	(* Reset Device by setting Error State  **********************)
	12:	
		IoDevReset(DEVICEID	:= DevId,RESET	:= TRUE );
		IF NOT IoDevReset.BUSY
		THEN
			IF IoDevReset.ERR THEN
				Busy										:= FALSE;
				Error										:= TRUE;
				ErrorId										:= IoDevReset.ERRID;
				ErrorText									:= CONCAT('IOF_DeviceReset Id: ',UDINT_TO_STRING(ErrorId));
				state 										:= 0;
			ELSE //Tr to                         					
				Error										:= FALSE;
				ErrorId										:= 0;
				ErrorText									:= '';
				DevResetDone 								:= TRUE;
				TON_TimeoutSetStatus(IN := FALSE);
				state 										:= 10;
			END_IF
		ELSE
			;
		END_IF
		
	(* Start to clear frame statistic **********************************)
	20: 
		FrameStatisticClearCRC(bExecute := Options.0);
		IF NOT FrameStatisticClearCRC.bBusy
		THEN
			IF FrameStatisticClearCRC.bError THEN
				Busy										:= FALSE;
				Error										:= TRUE;
				ErrorId										:= FrameStatisticClearCRC.nErrId;
				ErrorText									:= CONCAT('FB_EcMasterFrameStatisticClearCRC Id: ',UDINT_TO_STRING(ErrorId));
				state 										:= 0;
			ELSE                
				state 										:= state + 1;
			END_IF
		END_IF		
	
	21: 
		FrameStatisticClearFrames(bExecute := Options.1);
		IF NOT FrameStatisticClearFrames.bBusy
		THEN
			IF FrameStatisticClearFrames.bError THEN
				Busy										:= FALSE;
				Error										:= TRUE;
				ErrorId										:= FrameStatisticClearFrames.nErrId;
				ErrorText									:= CONCAT('FB_EcMasterFrameStatisticClearFrames Id: ',UDINT_TO_STRING(ErrorId));
				state 										:= 0;
			ELSE                
				state 										:= state + 1;
			END_IF
		END_IF	

	22: 
		FrameStatisticClearTxRxErr(bExecute := Options.2);
		IF NOT FrameStatisticClearTxRxErr.bBusy
		THEN
			IF FrameStatisticClearTxRxErr.bError THEN
				Busy										:= FALSE;
				Error										:= TRUE;
				ErrorId										:= FrameStatisticClearTxRxErr.nErrId;
				ErrorText									:= CONCAT('FB_EcMasterFrameStatisticClearTxRxErr Id: ',UDINT_TO_STRING(ErrorId));
				state 										:= 0;
			ELSE                
				Busy										:= FALSE;
				Done										:= TRUE;
				state 										:= 0;
			END_IF
		END_IF	
		
	ELSE
		;
	END_CASE
                										
(*********************************************************************)

{attribute 'monitoring' := 'call'}
PROPERTY PUBLIC optClearCRCErrorCounter : BOOL
GET
optClearCRCErrorCounter := Options.0;
END_GET
SET
Options.0 := optClearCRCErrorCounter;
END_SET
END_PROPERTY

{attribute 'monitoring' := 'call'}
PROPERTY PUBLIC optClearLostFramesCounter : BOOL
GET
optClearLostFramesCounter := Options.1;
END_GET
SET
Options.1 := optClearLostFramesCounter;
END_SET
END_PROPERTY

{attribute 'monitoring' := 'call'}
PROPERTY PUBLIC optClearTCRXErrCounter : BOOL
GET
optClearTCRXErrCounter := Options.2;
END_GET
SET
Options.2 := optClearTCRXErrCounter;
END_SET
END_PROPERTY

{attribute 'monitoring' := 'call'}
PROPERTY PUBLIC optForceDevReset : BOOL
GET
optForceDevReset := Options.7;
END_GET
SET
Options.7 := optForceDevReset;
END_SET
END_PROPERTY

END_FUNCTION_BLOCK

// POUs/Fieldbus/EtherCAT/_Components/EcSlavesDiag
{attribute 'no_check'}
{attribute 'enable_dynamic_creation'}
FUNCTION_BLOCK EcSlavesDiag EXTENDS FbBase
VAR CONSTANT
	SLAVE_ADDR_OFFSET										:	UINT := 1000;
	DEL_SSTATE_CHANGED										:	 TIME := T#2S;
END_VAR
VAR_OUTPUT CONSTANT         								
	MIN_SLAVES												: 	UINT := 1;
	MAX_SLAVES												: 	UINT := PARAM.ETHERCAT_DIAG_MAX_SLAVES;	//EC_MAX_SLAVES = 65535 Slaves;
	
{attribute 'displaymode':='binary'}
	OPTION_READ_SCAN_SLAVES									:	BYTE := 2#0000_0001; //Read scanned slaves identity and link State
{attribute 'displaymode':='binary'}
	OPTION_SORT_INFO_DATA									:	BYTE := 2#0000_0010; //Sort list of slaves InfoData according to scanned/physical sequence
{attribute 'displaymode':='binary'}
	OPTION_UPDATE_TOPO_DATA									:	BYTE := 2#0000_0100; //Read topology data, helpful if hot connect groups are configured
{attribute 'displaymode':='binary'}
	OPTION_UPDATE_CONFIG_DATA								:	BYTE := 2#0000_1000; //Read info slave data with with every execution	
END_VAR           
VAR_INPUT
	MasterAmsNetId											:	T_AmsNetId;
{attribute 'displaymode':='binary'}
	Options													:	BYTE := 0;
END_VAR
VAR_OUTPUT         
	NoOfSlaves												:	UINT;			//shows number of configured 
	NoOfSlavesNOK											:	UINT;  			//Shows number of slaves not in OP or with CRC error etc
	NoOfHCGroups											:	UINT;  			//Shows number of hot connect groups
	NoOfHCSlaves											:	UINT;  			//Shows number of slave in a hot connect group
	InfoData												:	ARRAY [MIN_SLAVES..MAX_SLAVES] OF EC_SLAVE_DIAG_INFO_DATA; //configures slaves			
	LastActiveSlave											:	EC_SLAVE_DIAG_INFO_DATA;	//shows last slave in OP connected to port A 
	FirstErrorSlave											:	EC_SLAVE_DIAG_INFO_DATA;	//shows first slave with an error
	InfoDataSorted											:	BOOL; //Info data list sorted according physical sequence vs. configured seq.
	InvalidVPRS												:	BOOL; //Invalid VPRS active
	ErrorText												:	STRING;		//shows error text of FB
	ExecutionTime											: 	TIME; //Total cycle time to execute the FB
END_VAR                     								         								
VAR                         								
(* Cache ********************************************************)               								
	pMemory													:	POINTER TO BYTE;
	SizeOfMemory											:	UDINT;
	MemNoOfSlaves											:	UINT;	
	ScannedSeqMixed											:	BOOL; //Scanned slave sequence is different to configured 

	pScannedSlaves											:	POINTER TO ARRAY [MIN_SLAVES..MAX_SLAVES] OF Tc2_EtherCAT.ST_EcSlaveScannedData;
	pConfigSlaves											:	POINTER TO ARRAY [MIN_SLAVES..MAX_SLAVES] OF Tc2_EtherCAT.ST_EcSlaveConfigData; 
	pSlavesState											:	POINTER TO ARRAY [MIN_SLAVES..MAX_SLAVES] OF Tc2_EtherCAT.ST_EcSlaveState;
	pSlavesStatusCode										:	POINTER TO ARRAY [MIN_SLAVES..MAX_SLAVES] OF DWORD;
	pTopologyData											:	POINTER TO ARRAY [MIN_SLAVES..MAX_SLAVES] OF Tc2_EtherCAT.ST_TopologyDataEx;
	
	StartTime												:	TIME;
	
(* timer ********************************************************)

(* trigger ********************************************************)

(* function-blocks *************************************************)
	EcGetSlaveCount											:	FB_EcGetSlaveCount := (tTimeout	:= T#60S);
	EcGetConfSlaves											:	FB_EcGetConfSlaves := (tTimeout	:= T#60S);
	EcGetScannedSlaves										:	FB_EcGetScannedSlaves := (tTimeout	:= T#60S);
	EcGetAllSlaveStateS										:	FB_EcGetAllSlaveStateS := (tTimeout	:= T#60S);
	EcGetAllSlaveCrcErrors									:	FB_EcGetAllSlaveCrcErrors := (tTimeout	:= T#60S);
	EcGetAllSlaveAbnormalStateChanges						:	FB_EcGetAllSlaveAbnormalStateChanges := (tTimeout	:= T#60S);	
	EcGetSlaveTopologyInfo									: 	FB_EcGetSlaveTopologyInfo := (tTimeout	:= T#60S);	
	
(* dummy **********************************************************)
	i,k,idx													:	UINT := 0;
	
END_VAR

	(* Check EtherCAT slaves status			V1	*)
	(********************************************)

(* Sequence *********************************)
	rtExecute(CLK := Execute);

	CASE State OF
	0:
		Busy 												:= FALSE;
		IF rtExecute.Q
		THEN //Clear data if FB is disabled or started
			Busy 											:= TRUE;
			Done											:= FALSE;
			Error											:= FALSE;
			Errorid											:= 0;
			ErrorText										:= '';	

		//	NoOfSlavesNIO									:= 0;	
			InvalidVPRS										:= FALSE;
			ScannedSeqMixed									:= FALSE;

			StartTime										:= TIME();
			ExecutionTime									:= T#0MS;
			
			EcGetSlaveCount(bExecute := FALSE,sNetId := MasterAmsNetId);
			EcGetConfSlaves(bExecute := FALSE,sNetId := MasterAmsNetId);
			EcGetSlaveTopologyInfo(bExecute := FALSE,sNetId := MasterAmsNetId);
			EcGetAllSlaveStates(bExecute := FALSE, sNetId := MasterAmsNetId);
			EcGetAllSlaveCrcErrors(bExecute := FALSE,sNetId := MasterAmsNetId);
			EcGetAllSlaveAbnormalStateChanges(bExecute := FALSE,sNetId := MasterAmsNetId);
			EcGetScannedSlaves(bExecute := FALSE,sNetId := MasterAmsNetId);
			
			MEMSET(ADR(LastActiveSlave),0,SIZEOF(LastActiveSlave));
			MEMSET(ADR(FirstErrorSlave),0,SIZEOF(FirstErrorSlave));
			
			IF NoOfSlaves = 0
			THEN
				State										:= 1;
			ELSIF Options.3 OR EcGetConfSlaves.nTotalSlaves = 0 OR InfoDataSorted
			THEN //Read config it not done or enabled
				State										:= 2;
			ELSIF Options.2 OR EcGetSlaveTopologyInfo.nSlaves = 0 OR InfoDataSorted
			THEN
				State										:= 10;
			ELSE
				State										:= 20;
			END_IF
		ELSIF NOT Execute
		THEN
			Done											:= FALSE;
			Error											:= FALSE;
			Errorid											:= 0;
			ErrorText										:= '';	
		END_IF
		IF StartTime > T#0MS AND ExecutionTime = T#0MS
		THEN
			ExecutionTime									:= TIME() - StartTime;
		END_IF
	
	(* Read no of configured slaves *********************************************************************)
	1:
		EcGetSlaveCount(bExecute := NoOfSlaves = 0);
		IF NOT EcGetSlaveCount.bBusy
		THEN
			IF EcGetSlaveCount.bError 
			THEN
				Busy										:= FALSE;
				Error										:= TRUE;
				ErrorId										:= EcGetSlaveCount.nErrId;
				ErrorText									:= CONCAT('EcGetSlaveCount Id: ',UDINT_TO_STRING(ErrorId));
				State 										:= 0;
			ELSIF EcGetSlaveCount.bExecute AND NoOfSlaves <> EcGetSlaveCount.nSlaves
			THEN
				NoOfSlaves									:= EcGetSlaveCount.nSlaves;					

				//Init Info Data 	
				MEMSET(ADR(InfoData),0,SIZEOF(InfoData));

				k 											:= NoOfSlaves + 1;
				//Set buffer lenght according to needed memory space
				EcGetConfSlaves.cbBufLen					:= SIZEOF(Tc2_EtherCAT.ST_EcSlaveConfigData) * k;
				EcGetScannedSlaves.cbBufLen					:= SIZEOF(Tc2_EtherCAT.ST_EcSlaveScannedData) * k;
				EcGetAllSlaveStates.cbBufLen				:= SIZEOF(Tc2_EtherCAT.ST_EcSlaveState) * k;
				EcGetAllSlaveCrcErrors.cbBufLen				:= SIZEOF(DWORD) * k;	
				EcGetSlaveTopologyInfo.cbBufLen				:= SIZEOF(Tc2_EtherCAT.ST_TopologyDataEx) * k;	
				EcGetAllSlaveAbnormalStateChanges.cbBufLen	:= EcGetAllSlaveCrcErrors.cbBufLen;						
					
				//Allocate dynamic buffer memory 
				IF Allocate(MAX(EcGetSlaveTopologyInfo.cbBufLen,MAX(MAX(EcGetConfSlaves.cbBufLen,EcGetAllSlaveCrcErrors.cbBufLen), MAX(EcGetScannedSlaves.cbBufLen,EcGetAllSlaveStateS.cbBufLen) )))
				THEN
					//Write buffer lenght per FB	
					pConfigSlaves							:= pMemory;
					pScannedSlaves							:= pMemory;
					pSlavesState							:= pMemory;
					pSlavesStatusCode						:= pMemory;	
					pTopologyData							:= pMemory;	
					
					State 									:= State + 1;			
				ELSE
					Busy									:= FALSE;
					Error									:= TRUE;
					ErrorId									:= E_AdsErr.DEVICE_NOMEMORY; //No memory
					ErrorText								:= CONCAT('EcSlavesDiag.allocate() Id: ',UDINT_TO_STRING(ErrorId));
					State 									:= 0;	
				END_IF

			ELSE
				State 										:= State + 1;
			END_IF
		ELSE
			;
		END_IF		
	
	
	(* Read slaves "configuration" ************************************************************************************************************)
	2:
		EcGetConfSlaves(bExecute := TRUE, pArrEcConfSlaveInfo := pConfigSlaves, cbBufLen := (* See State 1 *) );
			
		IF NOT EcGetConfSlaves.bBusy
		THEN
			IF EcGetConfSlaves.bError 
			THEN
				Busy										:= FALSE;
				Error										:= TRUE;
				ErrorId										:= EcGetConfSlaves.nErrorId;
				ErrorText									:= CONCAT('FB_EcGetConfSlaves Id: ',UDINT_TO_STRING(ErrorId));
				State										:= 0;     
					
			ELSIF EcGetConfSlaves.nSlaves > MAX_SLAVES
			THEN
				Busy										:= FALSE;
				Error										:= TRUE;
				ErrorId										:= E_AdsErr.DEVICE_INVALIDSIZE  ;
				ErrorText									:= CONCAT('No of config slaves > PARAM.ETHERCAT_MASTER_DIAG_MAX_SLAVES, please update value to ', TO_STRING(EcGetConfSlaves.nSlaves));
				State										:= 0;  					
			ELSE
				State 										:= State + 1;
			END_IF
		END_IF	
		
		
	3: //Fill structure	
		k													:= MIN(EcGetConfSlaves.nSlaves, NoOfSlaves);
		FOR i := MIN_SLAVES TO k DO
			InfoData[i].Addr								:= pConfigSlaves^[i].nAddr;
			InfoData[i].ConfigType							:= pConfigSlaves^[i].sType; 
		//	InfoData[i].DevType								:= pConfigSlaves^[i].nDevType;
			InfoData[i].ConfigName							:= DELETE(pConfigSlaves^[i].sName, LEN(InfoData[i].ConfigType) + 3 , FIND(pConfigSlaves^[i].sName,InfoData[i].ConfigType) - 1); //Delete type if in brakets 	
			InfoData[i].ConfigTypeIdentity					:= F_ConvProductCodeToString(pConfigSlaves^[i].stSlaveIdentity);
			InfoData[i].ConfigIdentity						:= pConfigSlaves^[i].stSlaveIdentity;
		//	InfoData[i].LinkState							:= pConfigSlaves^[i].nLinkStatus; see read slaves state					
		END_FOR
		
		State 												:= SEL(Options.2 OR EcGetSlaveTopologyInfo.nSlaves = 0 OR InfoDataSorted, 20, 10);	
		
	(* Read slaves "topology" information *******************************************************************************************************)
	10:
		EcGetSlaveTopologyInfo(bExecute := NoOfSlaves > 0 , sNetId	:= MasterAmsNetId,  pAddrBuf := pTopologyData,  cbBufLen	:= (* See State 1 *));
		IF NOT EcGetSlaveTopologyInfo.bBusy
		THEN
			IF EcGetSlaveTopologyInfo.bError 
			THEN
				Busy										:= FALSE;
				Error										:= TRUE;
				ErrorId										:= EcGetSlaveTopologyInfo.nErrId;
				ErrorText									:= CONCAT('EcGetSlaveTopologyInfo Id: ',UDINT_TO_STRING(ErrorId));
				State 										:= 0;
			ELSIF EcGetSlaveTopologyInfo.nSlaves > MAX_SLAVES
			THEN
				Busy										:= FALSE;
				Error										:= TRUE;
				ErrorId										:= E_AdsErr.DEVICE_INVALIDSIZE  ;
				ErrorText									:= CONCAT('No of scanned slaves > PARAM.ETHERCAT_MASTER_DIAG_MAX_SLAVES, please update value to ', TO_STRING(EcGetScannedSlaves.nSlaves));
				State										:= 0;  	
			ELSE
				State 										:= State + 1;
			END_IF
		ELSE
			;
		END_IF	

	11:	//Fill structure		
		NoOfHCGroups										:= 0;
		NoOfHCSlaves										:= 0;
		k													:= MIN(EcGetSlaveTopologyInfo.nSlaves, NoOfSlaves);
		FOR i := MIN_SLAVES TO k DO                 		
			InfoData[i].TopoOwnPhysicalAddr					:= pTopologyData^[i].nOwnPhysicalAddr; 
			InfoData[i].TopologyStatus						:= pTopologyData^[i].nStatusBits;
			InfoData[i].HCSlaveCountCfg  					:= pTopologyData^[i].nHCSlaveCountCfg;
			InfoData[i].HCSlaveCountAct  					:= pTopologyData^[i].nHCSlaveCountAct;
			InfoData[i].AutoIncAddr   						:= pTopologyData^[i].nOwnAutoIncAddr;
			InfoData[i].PhysicalPortAddr    				:= pTopologyData^[i].stPhysicalAddr;
			InfoData[i].AutoIncPortAddr    					:= pTopologyData^[i].stAutoIncAddr;
			                                        		
			InfoData[i].HotConnectNodeStart 				:= InfoData[i].TopologyStatus.3;
			InfoData[i].HotConnectSlave 					:= InfoData[i].TopologyStatus.4;
                                                    		
			NoOfHCGroups									:= SEL(InfoData[i].HotConnectNodeStart , NoOfHCGroups, NoOfHCGroups + 1);
			NoOfHCSlaves									:= SEL(InfoData[i].HotConnectSlave , NoOfHCSlaves, NoOfHCSlaves + 1);
			                                        	
		END_FOR				                        	
		State 												:= 20;
		
	(* Read slaves "EtherCAT State and link state" ***************************************************************************************)
	20	:
		EcGetAllSlaveStateS(bExecute := NoOfSlaves > 0, pStateBuf:=  pSlavesState, cbBufLen	:= (* See State 1 *));
					
		IF NOT EcGetAllSlaveStateS.bBusy
		THEN
			IF EcGetAllSlaveStateS.bError 
			THEN
				Busy										:= FALSE;
				Error										:= TRUE;
				ErrorId										:= EcGetAllSlaveStateS.nErrId;
				ErrorText									:= CONCAT('FB_EcGetAllSlaveStates Id: ',UDINT_TO_STRING(ErrorId));
				State 										:= 0;
			ELSE
				k											:= MIN(EcGetAllSlaveStateS.nSlaves, NoOfSlaves);
				FOR i := MIN_SLAVES TO k DO
					InfoData[i].LinkState					:= pSlavesState^[i].linkState;
					InfoData[i].DevState					:= pSlavesState^[i].deviceState;
					InfoData[i].DevStateText				:= F_ConvSlaveStateToString(pSlavesState^[i]);
					InfoData[i].DevStateBits				:= F_ConvSlaveStateToBitsEx(pSlavesState^[i]);	
					InfoData[i].ErrorIdentCode.0			:= InfoData[i].DevStateBits.bInvVPRS; //Wrong slave
					IF InfoData[i].ErrorIdentCode.0 THEN InvalidVPRS := TRUE; END_IF
					InfoData[i].ErrorIdentCode.1			:= NOT InfoData[i].ErrorIdentCode.0 AND NOT InfoData[i].DevStateBits.bOp AND_THEN(NOT InfoData[i].HotConnectSlave OR NOT InfoData[i].DevStateBits.bInit); //Wrong State
				END_FOR	

				State 										:= State + 1;
			END_IF
		ELSE
			;
		END_IF	
		
	(* Get all slaves "CRC counter" ********************************************************************)
	21:	
		EcGetAllSlaveCrcErrors(bExecute := NoOfSlaves > 0, sNetId	:= MasterAmsNetId,  pCrcErrorBuf:= pSlavesStatusCode,  cbBufLen	:= (* See State 1 *));
		IF NOT EcGetAllSlaveCrcErrors.bBusy
		THEN
			IF EcGetAllSlaveCrcErrors.bError 
			THEN
				Busy										:= FALSE;
				Error										:= TRUE;
				ErrorId										:= EcGetAllSlaveStateS.nErrId;
				ErrorText									:= CONCAT('FB_EcGetAllSlaveCrcErrors Id: ',UDINT_TO_STRING(ErrorId));
				State 										:= 0;
			ELSE
				k											:= MIN(EcGetAllSlaveCrcErrors.nSlaves, NoOfSlaves);
				FOR i := MIN_SLAVES TO k DO
					InfoData[i].ErrorIdentCode.2			:= InfoData[i].CntOfCRCErrors <> pSlavesStatusCode^[i] AND pSlavesStatusCode^[i] > 0; //CRC error increased
					InfoData[i].CntOfCRCErrors				:= pSlavesStatusCode^[i];				
				END_FOR				
				
				State 										:= State + 1;
			END_IF
		ELSE
			;
		END_IF
		
	(* Get all slaves "no of abnormal state change" *****************************************************************************)
	22:	
		EcGetAllSlaveAbnormalStateChanges(bExecute := NoOfSlaves > 0, sNetId	:= MasterAmsNetId,  pAddrBuf := pSlavesStatusCode,  cbBufLen	:= (* See State 1 *));
		IF NOT EcGetAllSlaveAbnormalStateChanges.bBusy
		THEN
			IF EcGetAllSlaveAbnormalStateChanges.bError 
			THEN
				Busy										:= FALSE;
				Error										:= TRUE;
				ErrorId										:= EcGetAllSlaveAbnormalStateChanges.nErrId;
				ErrorText									:= CONCAT('FB_EcGetAllSlaveAbnormalStateChanges Id: ',UDINT_TO_STRING(ErrorId));
				State 										:= 0;
			ELSE
				k											:= MIN(EcGetAllSlaveAbnormalStateChanges.nSlaves, NoOfSlaves);
				FOR i := MIN_SLAVES TO k DO
					InfoData[i].ErrorIdentCode.3			:= InfoData[i].NoOfAbnormalStateChanges <> pSlavesStatusCode^[i] AND pSlavesStatusCode^[i] > 0; //Abnormal State change increased
					InfoData[i].NoOfAbnormalStateChanges	:= pSlavesStatusCode^[i];	
				END_FOR				
				
				State 										:= SEL(Options.0 OR EcGetScannedSlaves.nSlaves = 0, 40, 30);
			END_IF
		ELSE
			;
		END_IF

	(* Start to read scanned slaves *************************************************************************)
	30:
		EcGetScannedSlaves(bExecute := TRUE, pArrEcScannedSlaveInfo  := pScannedSlaves, cbBufLen := (* See State 1 *));
			
		IF NOT EcGetScannedSlaves.bBusy
		THEN
			IF EcGetScannedSlaves.bError 
				AND EcGetScannedSlaves.nErrorId <> 1817 //device has a timeout -> not error if no slave is connected 
			THEN
				Busy										:= FALSE;
				Error										:= TRUE;
				ErrorId										:= EcGetScannedSlaves.nErrorId;
				ErrorText									:= CONCAT('FB_EcGetScannedSlaves Id: ',UDINT_TO_STRING(ErrorId));
				State										:= 0;     

			ELSIF EcGetScannedSlaves.nSlaves > MAX_SLAVES
			THEN
				Busy										:= FALSE;
				Error										:= TRUE;
				ErrorId										:= E_AdsErr.DEVICE_INVALIDSIZE  ;
				ErrorText									:= CONCAT('No of scanned slaves > PARAM.ETHERCAT_MASTER_DIAG_MAX_SLAVES, please update value to ', TO_STRING(EcGetScannedSlaves.nSlaves));
				State										:= 0;  			
			
			ELSE	
				FOR i := MIN_SLAVES TO NoOfSlaves 
				DO					
					InfoData[i].ScannedTypeIdentity			:= '<not present>';
					MEMSET(ADR(InfoData[i].ScannedIdentity),0,SIZEOF(InfoData[i].ScannedIdentity));								
					InfoData[i].DataLinkStatusReg			:= 0;	
					InfoData[i].ScannedSeq					:= 0;						
				END_FOR
				State 										:= SEL(EcGetScannedSlaves.nSlaves = 0, State + 1, 40);
			END_IF
		END_IF
		
	31: //Fill structure
		k													:= MIN(EcGetScannedSlaves.nSlaves,NoOfSlaves); //No of scanned slaves
		idx													:= 0;
		ScannedSeqMixed										:= FALSE;
		FOR i := MIN_SLAVES TO NoOfSlaves DO		
			IF i <= EcGetScannedSlaves.nSlaves
			THEN
				idx											:= SEL(pScannedSlaves^[i].nAddr > SLAVE_ADDR_OFFSET, idx + 1 ,pScannedSlaves^[i].nAddr - SLAVE_ADDR_OFFSET);
				InfoData[idx].ScannedTypeIdentity			:= F_ConvProductCodeToString(pScannedSlaves^[i].stSlaveIdentity);
				InfoData[idx].ScannedIdentity				:= pScannedSlaves^[i].stSlaveIdentity;				
				InfoData[idx].DataLinkStatusReg				:= pScannedSlaves^[i].ndlStatusReg;		
				InfoData[idx].ScannedSeq					:= i;	
				ScannedSeqMixed								:= i <> idx OR ScannedSeqMixed;
			ELSE
				EXIT;
			END_IF
		
		END_FOR
		
		State 												:= 40;
		
	(* Search for error slaves **************************************************************************)
	40:
		k													:= EcGetScannedSlaves.nSlaves + 1; 
		NoOfSlavesNOK										:= 0;
		FOR i := MIN_SLAVES TO NoOfSlaves				
		DO
			//Fill PhysicalSeq number of missed slaves for possible sorting
			IF ScannedSeqMixed AND Options.1
			THEN
				IF InfoData[i].ScannedSeq = 0
				THEN 										
					InfoData[i].ScannedSeq 					:= k;
					k										:= k + 1;
				END_IF
			END_IF
		
			//Search for first slave with error
			IF InfoData[i].ErrorIdentCode <> 0
			THEN
				NoOfSlavesNOK								:= NoOfSlavesNOK + 1;
				IF FirstErrorSlave.Addr = 0
				THEN
					FirstErrorSlave 						:= InfoData[i]; 					
					IF i - 1 > 0
					THEN
						LastActiveSlave 					:= InfoData[i - 1];
					END_IF
				END_IF						
			END_IF
		END_FOR   	
	
		IF ScannedSeqMixed AND Options.1
		THEN
			InfoDataSorted									:= TRUE;
			State											:= State + 1;
		ELSE
			InfoDataSorted									:= FALSE;
			Busy											:= FALSE;
			Done											:= TRUE;
			State											:= 0;   
		END_IF
	
	(* Sort InfoData list if sequence is mixed and option selected **************************************************************************)	
	41: 
		IF sortList()
		THEN
			Busy											:= FALSE;
			Done											:= TRUE;
			State											:= 0;   
		ELSE
			Busy											:= FALSE;
			Error											:= TRUE;
			ErrorId											:= E_AdsErr.DEVICE_INVALIDDATA  ; //Invalid data
			ErrorText										:= 'Error sorting InfoData list ';
			State											:= 0;  			
		END_IF	
 
	ELSE
		;
	END_CASE

(***********************************************************************)

METHOD PROTECTED FINAL allocate : BOOL
VAR_INPUT 
	MemSize													:	UDINT;
END_VAR
VAR
END_VAR
IF MemSize = 0
THEN
	allocate												:= FALSE;	
ELSIF pMemory = 0 
THEN
	pMemory													:= __NEW(BYTE,MemSize );
	SizeOfMemory											:= MemSize;
	IF PARAM.ENABLE_DEBUG_MSG_DYNAMIC_MEM_ALLOCATION
	THEN
		AdsLogHint('EngineeringToolbox | FB EcSlavesDiag | An instance allocated %s bytes from the dynamic memory of the ADS router memory pool', TO_STRING(MemSize));
	END_IF
	Allocate												:= TRUE;	
ELSIF MemSize > SizeOfMemory
THEN//Size increased, allocate new memory
	__DELETE(pMemory);  //Delete reference to old memory
	
	pMemory													:= __NEW(BYTE,MemSize );
	SizeOfMemory											:= MemSize;
	IF PARAM.ENABLE_DEBUG_MSG_DYNAMIC_MEM_ALLOCATION
	THEN
		AdsLogWarn('EngineeringToolbox | FB EcSlavesDiag | No of slaves increased and one instance allocated additional %s bytes from the dynamic memory of the ADS router memory pool', TO_STRING(MemSize));
	END_IF

	Allocate												:= TRUE;
ELSE
	Allocate												:= FALSE;
END_IF
END_METHOD

METHOD FB_exit : BOOL
VAR_INPUT
	bInCopyCode : BOOL; // if TRUE, the exit method is called for exiting an instance that is copied afterwards (online change).
END_VAR
IF NOT bInCopyCode AND pMemory <> 0
THEN //Release memory in case the PLC stopps
	__DELETE(pMemory);
	SizeOfMemory								:= 0;
END_IF
END_METHOD

{attribute 'monitoring' := 'call'}
PROPERTY PUBLIC optReadScannedSlaves : bool
GET
optReadScannedSlaves := Options.0;
END_GET
SET
OPtions.0 := optReadScannedSlaves;
END_SET
END_PROPERTY

{attribute 'monitoring' := 'call'}
PROPERTY PUBLIC optSortInfoData : bool
GET
optSortInfoData := Options.2;
END_GET
SET
OPtions.2 := optSortInfoData;
END_SET
END_PROPERTY

{attribute 'monitoring' := 'call'}
PROPERTY PUBLIC optUpdateConfigData : bool
GET
optUpdateConfigData := Options.3;
END_GET
SET
OPtions.3 := optUpdateConfigData;
END_SET
END_PROPERTY

{attribute 'monitoring' := 'call'}
PROPERTY PUBLIC optUpdateTopoData : bool
GET
optReadScannedSlaves := Options.1;
END_GET
SET
OPtions.1 := optReadScannedSlaves;
END_SET
END_PROPERTY

METHOD INTERNAL sortList : BOOL
VAR_INPUT
END_VAR
VAR
	SlaveInfoData1											:	EC_SLAVE_DIAG_INFO_DATA;
	SlaveInfoData2											:	EC_SLAVE_DIAG_INFO_DATA;
END_VAR
	sortList												:= TRUE;
	
	i														:= MIN_SLAVES;
	WHILE i <= NoOfSlaves OR SlaveInfoData1.ScannedSeq <> 0 
	DO
		IF SlaveInfoData1.ScannedSeq > 0
		THEN
			IF SlaveInfoData1.ScannedSeq > NoOfSlaves
			THEN //Error seq no
				sortList									:= FALSE;
				EXIT;
			ELSE
				SlaveInfoData2 								:= InfoData[SlaveInfoData1.ScannedSeq]; //Backup target
				InfoData[SlaveInfoData1.ScannedSeq].ScannedSeq	:= 0; //Mark as copied				
				InfoData[SlaveInfoData1.ScannedSeq]			:= SlaveInfoData1; //Copy from cache into target	
				SlaveInfoData1								:= SlaveInfoData2; //Write backed up data into cache
			END_IF

		ELSIF InfoData[i].ScannedSeq > 0 AND InfoData[i].ScannedSeq <> i
		THEN
			//Put target into cache
			SlaveInfoData1									:= InfoData[InfoData[i].ScannedSeq];
			InfoData[InfoData[i].ScannedSeq]				:= InfoData[i];		
			InfoData[i].ScannedSeq							:= 0; //Mark as copied
		ELSE
			;				
		END_IF   
		i													:= i + 1;
	END_WHILE;
END_METHOD

END_FUNCTION_BLOCK

// POUs/Fieldbus/EtherCAT/_Components/EcSlaveSupervisor
{attribute 'no_check'}
(* Set EtherCAT state(ReqState <> 0) or read state and CRC error counter of EtherCAT slave *)
FUNCTION_BLOCK EcSlaveSupervisor Extends FbBase
VAR_INPUT
	EcMasterAmsNetId										:	T_AmsNetId;
	SlaveAddr												: 	UINT; 		//-> Slave Port number!
{attribute 'displaymode':='hex'}
	ReqState												:	WORD := 0; (* 	EC_DEVICE_STATE_INIT		:BYTE 	:=16#01;
																				EC_DEVICE_STATE_PREOP		:BYTE 	:=16#02;
																				EC_DEVICE_STATE_BOOTSTRAP	:BYTE 	:=16#03;
																				EC_DEVICE_STATE_SAFEOP		:BYTE 	:=16#04;
																				EC_DEVICE_STATE_OP			:BYTE 	:=16#08; *)																				
END_VAR                     							
VAR_OUTPUT                  							
{attribute 'displaymode':='hex'}
	CurrState												: 	BYTE;	(* Shows current state 																					
																				EC_DEVICE_STATE_INIT		:BYTE 	:=16#01;
																				EC_DEVICE_STATE_PREOP		:BYTE 	:=16#02;
																				EC_DEVICE_STATE_BOOTSTRAP	:BYTE 	:=16#03;
																				EC_DEVICE_STATE_SAFEOP		:BYTE 	:=16#04;
																				EC_DEVICE_STATE_OP			:BYTE 	:=16#08; *)
{attribute 'displaymode':='hex'}
	linkState												: 	BYTE;	(* Shows state of link
																				EC_LINK_STATE_OK :BYTE :=16#00;
																				EC_LINK_STATE_NOT_PRESENT :BYTE :=16#01;
																				EC_LINK_STATE_LINK_WITHOUT_COMM :BYTE :=16#02;
																				EC_LINK_STATE_MISSING_LINK :BYTE :=16#04;
																				EC_LINK_STATE_ADDITIONAL_LINK :BYTE :=16#08;
																				EC_LINK_STATE_PORT_A :BYTE :=16#10;
																				EC_LINK_STATE_PORT_B :BYTE :=16#20;
																				EC_LINK_STATE_PORT_C :BYTE :=16#40;
																				EC_LINK_STATE_PORT_D :BYTE :=16#80; *)
																				
	ReqStateOK												:	BOOL;		//Requested state of slave is OK
	StateBits												:	ST_EcSlaveStateBitsEx;
	StateText												:	STRING(80);	//State as text
	CrcError    											:    ST_EcCrcErrorEx; (*Crc error of the EtherCAT slave device*)
END_VAR                 								
VAR                     								
	TON_GetStateTrig										:	TON;
	SetSlaveState											:	FB_EcSetSlaveSTATE := (tTimeout := DEFAULT_ADS_TIMEOUT);
	GetSlaveState											:	FB_EcGetSlaveSTATE := (tTimeout := DEFAULT_ADS_TIMEOUT);
	GetSlaveCrcErrorEx 										:	FB_EcGetSlaveCrcErrorEx  := (tTimeout := DEFAULT_ADS_TIMEOUT);
	MemReqState												:	WORD;
	ErrorText												:	STRING(40);
END_VAR

	(* Set EtherCAT state(ReqState <> 0) or read state and CRC error counter of EtherCAT slave *)
	(*******************************************************************************************)

(* Process ******************************************************)
	rtExecute(CLK := Execute);

	CASE state OF
	(* cyclic reading of state ***********************************)
	0:
		Busy 												:= FALSE;

		IF rtExecute.Q 
		THEN
			Busy 											:= TRUE;
			Done											:= FALSE;
			Error											:= FALSE;
			ErrorID											:= 0;
			Errortext										:= '';
			CurrState										:= 0;
			linkState										:= 0;
			ReqStateOK										:= FALSE;
			MEMSET(ADR(StateBits),0,SIZEOF(StateBits));
			MEMSET(ADR(CrcError),0,SIZEOF(CrcError));	
			StateText										:= '';
	
			SetSlaveSTATE(bExecute := FALSE, sNetId:= EcMasterAmsNetId,nSlaveAddr:= SlaveAddr);
			GetSlaveSTATE(bExecute := FALSE,sNetId:= EcMasterAmsNetId,nSlaveAddr:= SlaveAddr);
			GetSlaveCrcErrorEx(bExecute := FALSE,sNetId:= EcMasterAmsNetId,nSlaveAddr:= SlaveAddr);

			IF(ReqState <> CurrState
				OR ReqState <> MemReqState)
				AND ReqState <> 0
			THEN
				SetSlaveState(bExecute:= TRUE,reqState:= ReqState);
				MemReqState 								:= ReqState;
				state 										:= 10;

			ELSE
				(* Start Reading State *)
				GetSlaveState(bExecute	:= TRUE);
				state 										:= 1;
			END_IF

		ELSIF NOT Execute 
		THEN
			Done 											:= FALSE;
			Error											:= FALSE;
			ErrorID											:= 0;
			ErrorText										:= '';
		END_IF

	(* Read Slave State **************************************)
	1:
		(* Work block *)
		GetSlaveState();

		IF NOT GetSlaveState.bBusy
		THEN
			IF GetSlaveState.bError THEN
				Busy										:= FALSE;
				Error										:= TRUE;
				ErrorId										:= GetSlaveState.nErrId;
				ErrorText									:= CONCAT('FB_EcGetSlaveSTATE Id: ',UDINT_TO_STRING(ErrorId));
				state 										:= 0;
			ELSE       
				ReqStateOK 									:= (ReqState = CurrState OR ReqState = 0);         					
				CurrState 									:= GetSlaveState.state.deviceState;
				linkState 									:= GetSlaveState.State.linkState;
				StateText 									:= F_ConvStateToString(GetSlaveState.State.deviceState);
			 	StateBits							 		:= F_ConvSlaveStateToBitsEx(GetSlaveState.state);
				state										:= state + 1;
			END_IF
			GetSlaveSTATE(bExecute := FALSE);
		ELSE
			;
		END_IF

	(* Read Slave CRC Error Counter  **************************************)		
	2: 
		(* Work block *)
		GetSlaveCrcErrorEx();

		IF NOT GetSlaveCrcErrorEx.bBusy
		THEN
			IF GetSlaveCrcErrorEx.bError THEN
				Busy										:= FALSE;
				Error										:= TRUE;
				ErrorId										:= GetSlaveCrcErrorEx.nErrId;
				ErrorText									:= CONCAT('FB_EcGetSlaveCrcErrorEx Id: ',UDINT_TO_STRING(ErrorId));
				state 										:= 0;
			ELSE       
				CrcError									:= 	GetSlaveCrcErrorEx.crcError;
				Done 										:= TRUE;
				Busy 										:= FALSE;
				state										:= 0;
			END_IF
			GetSlaveCrcErrorEx(bExecute := FALSE);
		ELSE
			;
		END_IF

	(* Set state  *****************************************)
	10:	
		SetSlaveState();  
		IF NOT SetSlaveState.bBusy
		THEN
			IF SetSlaveState.bError 
			THEN             	
				Busy										:= FALSE;
				Error										:= TRUE;
				ErrorId										:= SetSlaveState.nErrId;
				ErrorText									:= CONCAT('FB_EcSetSlaveSTATE Id: ',UDINT_TO_STRING(ErrorId));
				state 										:= 0;
			ELSIF SetSlaveState.CurrState.deviceState = MemReqState 
			THEN
				ReqStateOK									:= TRUE;
				Busy 										:= FALSE;
				Done 										:= TRUE;	
				state 										:= 0;
			ELSE                    				
				Busy										:= FALSE;		
				Error										:= TRUE;
				ErrorId										:= E_AdsErr.DEVICE_ABORTED;
				ErrorText									:= 'SetSlaveState DEVICESTATE <> ReqState';
				state	 									:= 0;
			END_IF         					
			CurrState 										:= SetSlaveState.currState.deviceState;
			linkState 										:= SetSlaveState.currState.linkState;
			StateText 										:= F_ConvStateToString(SetSlaveState.currState.deviceState);
			StateBits							 			:= F_ConvSlaveStateToBitsEx(SetSlaveState.currState);
			SetSlaveState(bExecute := FALSE);              						
		END_IF                      						
	END_CASE


(*********************************************************************)

END_FUNCTION_BLOCK

// POUs/Fieldbus/EtherCAT/EcCoEReadNewestDiagMsg
{attribute 'no_check'}
//Read EtherCAT diag newest message from EtherCAT slave via CoE
FUNCTION_BLOCK EcCoEReadNewestDiagMsg EXTENDS fbBase      
VAR CONSTANT
	{attribute 'displaymode':='hexadecimal'} 
	COE_DIAG_OBJECT											: WORD := 16#10F3;
END_VAR                  						
VAR_INPUT                           						
	AdsAddr													: 	AMSADDR; //Terminal AMS Net Addr.
	Timeout													:	TIME := DEFAULT_ADS_TIMEOUT;
END_VAR
VAR_IN_OUT
END_VAR
VAR_OUTPUT
	{attribute 'displaymode':='hexadecimal'}
	Message													: ARRAY[0..63] OF BYTE; //Index A010 with a lenght of 27 or 32/64 bytes subindex
	{attribute 'displaymode':='hexadecimal'}
	DiagCode												: UDINT; // first 4 bytes of message

	{attribute 'displaymode':='hexadecimal'}
	TextId													: UINT; //xyzz -> X =Type | y = Source | zz = Message ID
	Timestamp												: T_DCTIME64;	

	MsgSeverity												: UINT; //Extracted from Flags ->  -> 0:Info | 1:Warning | 2:Error 
	MsgTimestampLocal										: BOOL; //Extracted from Flags bit 4
	MsgNoOfParameter										: UINT; //Extracted from Flags 

	{attribute 'displaymode':='hexadecimal'}
	MsgType													: UINT; //Extracted from TextId -> 0=SystemInfo | 1:Info | 2:reserved | 4:Warning | 8:Error
	MsgSource												: UINT; //Extracted from TextId -> 0:System | 1:General | 2:Communication | 3:Encoder | 4:Drive | 5:Inputs | 6:IO | 7:Reserved 
	{attribute 'displaymode':='hexadecimal'}
	MsgId													: UINT; //Extracted from TextId 
END_VAR                             						
VAR

END_VAR
VAR
(* Cache *********************************************************************)	
	{attribute 'displaymode':='hexadecimal'}
	SubIndexNewestMessage									: BYTE;

	{attribute 'displaymode':='hexadecimal'}
	Flags													: UINT; //Info (0) Warning (1) or Error (2)
(* Timer ********************************************************************************)
  	
(* Trigger ******************************************************************************)


(* Function blocks ****************************************************************************)
	CoERead													: FB_EcCoeSdoReadEx;

(* Dummy Speicher **********************************************************)
	
END_VAR

	(* Read newest diag message															*)
	(************************************************************************************)

(* Sequence *****************************************************************)
	rtExecute(CLK := Execute);
	CASE state OF
	0: // Read subindex of the newest diagnosis message		
		busy												:= FALSE;
		IF rtExecute.Q
		THEN
			Busy											:= TRUE;
			Done											:= FALSE;
			Error											:= FALSE;
			ErrorId											:= 0;
			CoERead(bExecute := FALSE, sNetId := F_CreateAmsNetId(nIds := AdsAddr.netId),  nSlaveAddr := AdsAddr.port, bCompleteAccess:= FALSE ,nIndex := COE_DIAG_OBJECT , tTimeout := Timeout);
			
			MEMSET(ADR(Message),0,SIZEOF(Message));
			DiagCode										:= 0;
			Flags											:= 0;
			TextId											:= 0;
			Timestamp										:= 0;
			MsgType											:= 0;
			MsgSource										:= 0;
			MsgId											:= 0;
			
			state											:= state + 1;
		ELSIF NOT Execute
		THEN
			Done											:= FALSE;
			Error											:= FALSE;
			ErrorId											:= 0;
		END_IF
	1: // read subindex of newest diagnosis message
		CoERead(
			bExecute	:= TRUE, //Diagnosis histroy object
			nSubIndex	:= 16#02, // subindex newest message
			pDstBuf		:= ADR(SubIndexNewestMessage), 
			cbBufLen	:= SIZEOF(SubIndexNewestMessage) );
				
		IF NOT CoERead.bBusy
		THEN
			IF CoERead.bError
			THEN
				Busy										:= FALSE;
				Error										:= TRUE;
				ErrorId										:= CoERead.nErrId;
				state										:= 0;
			ELSE		
				state										:= state + 1;
			END_IF			
			CoERead(bExecute := FALSE );				
		END_IF
		
	2: // Read newest diagnosis messages from sub index
		CoERead(
			bExecute	:= TRUE, 
			nSubIndex	:= SubIndexNewestMessage, 
			pDstBuf		:= ADR(Message), 
			cbBufLen	:= SIZEOF(Message));
			
		IF NOT CoERead.bBusy
		THEN
			IF CoERead.bError
			THEN
				Busy										:= FALSE;
				Error										:= TRUE;
				ErrorId										:= CoERead.nErrId;
				state										:= 0;				
			ELSE // Copy certain byte arrays of the diagnosis messages to lcoal variables
				
				MEMCPY(ADR(DiagCode), ADR(Message[1]), 4); 		// copy 4 bytes of diag code data
				MEMCPY(ADR(Flags), ADR(Message[5]), 2); 		// copy 2 bytes of flag data
				MEMCPY(ADR(TextID),ADR(Message[7]), 2);			// copy 2 bytes of TextId data
				MEMCPY(ADR(Timestamp),ADR(Message[9]), 8);		// copy 8 bytes of 64bit DC time
				
				MsgType										:= SHR(TextId AND 16#F000, 12);
				MsgSource									:= SHR(TextId AND 16#0F00, 8);
				MsgId										:= TextId AND 16#00FF;
				MsgSeverity									:= Message[5] AND 2#0000_1111;
				MsgTimestampLocal							:= Message[5].4;
				MsgNoOfParameter							:= Message[6];
				
				Done										:= TRUE;
				state										:= 0;			
			END_IF
			CoERead(bExecute := False);		
		END_IF
	END_CASE


(******************************************************************************)

{attribute 'monitoring' := 'call'}
PROPERTY PUBLIC msgSevyIsError : BOOL
GET
msgSevyIsError := MsgSeverity = 2;
END_GET
END_PROPERTY

{attribute 'monitoring' := 'call'}
PROPERTY PUBLIC msgSevyIsInfo : BOOL
GET
msgSevyIsInfo := MsgSeverity = 0;
END_GET
END_PROPERTY

{attribute 'monitoring' := 'call'}
PROPERTY PUBLIC msgSevyIsWarning : BOOL
GET
msgSevyIsWarning := MsgSeverity = 1;
END_GET
END_PROPERTY

END_FUNCTION_BLOCK

// POUs/System/SystemInfo
{attribute 'no_check'}
//Provides all information of PlcAppSystemInfo plus addtional infos like time stamps from various source and in different formats
//
//PlcAppSystemInfo -> https://infosys.beckhoff.com/english.php?content=../content/1033/globaldatatypes/9007199969559691.html&id=7934476013631172214
//TwimCAT time sources -> https://infosys.beckhoff.com/english.php?content=../content/1033/ethercatsystem/2469114379.html&id=
//
FUNCTION_BLOCK SystemInfo
VAR_OUTPUT CONSTANT
{attribute 'displaymode':='binary'}
	OPTION_US_DATE_FORMAT									:	BYTE := 2#0000_0001; //Enable US date format in time stamp - mm/dd/yy
{attribute 'displaymode':='binary'}
	OPTION_US_TIME_FORMAT									:	BYTE := 2#0000_0010; //Enable time in US format - AM/PM vs 24h
{attribute 'displaymode':='binary'} 
	OPTION_TIME_STR_ADD_MS									:	BYTE := 2#0000_0100; //Add ms to time string 
{attribute 'displaymode':='binary'} 
	OPTION_DISABLE_DEV_IDENT								:	BYTE := 2#0000_1000; //Disable to read device identification during boot up (Call FB_GetDeviceIdentificationEx)
END_VAR                     								
VAR_INPUT                   						
	Enable													:	BOOL := TRUE; //Enable function block
	ResetTrig												:	BOOL := FALSE; //Reset Old boot data fault signal
	RtcSyncCylce											:	DWORD := 60; //in seconds - see documentation for "FB_LocalSystemTime"
	KeepOutputsOnBP 										: 	BOOL := FALSE; //The flag can be set to avoid that the outputs are zero-filled if a breakpoint is reached. The task keeps running. Only the execution of PLC code is interrupted.
{attribute 'displaymode':='binary'}
	Options													:	BYTE := 2#0000_0000; //option constants are alreay predefined, so they can accordingly be passed symbolically to the block 
	DateStrSeperator										:	STRING(1) := '/';
END_VAR
VAR_OUTPUT
//PlcAppSystemInfo and cycle time inforamtion from caller task 
	ObjId													: 	OTCID; //Object ID of the PLC project instance
	AdsPort 												: 	UINT; //ADS port of PLC application 
	TComSrvPtr 												: 	ITComObjectServer; // Pointer to TcCOM Object Server 
	AppName													: 	STRING(63); //TwinCAT generated name containing the port number. 
	ProjectName 											: 	STRING(63); //The name of the PLC project. 
	AppTimestampDT											:	DT; //Date and time of application start 
	AppTimestamp											:	STRING(25);	//Date and time of application start in string format
	TaskIndex												:	INT ; //Task index of SysInfo caller
	TaskCnt													: 	UDINT; //The number of tasks in the actual runtime system
	
	Flags 													: 	DWORD; //Boot flags
	LicensesPending 										: 	BOOL;
	BSODOccured 											: 	BOOL;										
	BootDataLoaded											: 	BOOL;//PERSISTENT variables: LOADED (without error)
	OldBootData												: 	BOOL; //PERSISTENT variables: INVALID (the back-up copy was loaded, since no valid data was present)
	NoBootDataLoaded										:	BOOL; //Error no boot data loaded
//	PersistentStatus 										: 	EPlcPersistentStatus;

	LoggedIn												:	BOOL;
	ShutdownInProgress 										: 	BOOL;	
	OnlineChangeCount										: 	UDINT; //The number of online changes made since the last complete download.
	OnlineChange											:	BOOL; //Online change count changed since last plc cycle

{attribute 'displaymode':='hex'}
	CpuCounter												:	ULINT;
	CycleTime         										: 	UDINT;//Cylce time read from PlcAppSystemInfo in multiples of 100 ns.
	CycleTimeNS         									: 	UDINT;//Cylce time in nanoseconds
	CycleTimeT       										: 	TIME; //Cycle time in time format
	CycleTimeLT       										: 	LTIME; //Cycle time in ltime format
	CycleTimeFloat											:	LREAL;//Cycle time in float format <s.ms>

	DevIdentValid											:	BOOL;
	pDevIdent												:	POINTER TO ST_DeviceIdentificationEx := ADR(InstGetDevIdent.stDevIdent);
	
//General	
	TimezoneId												: 	E_TimeZoneID;
	TimeZoneInfo											:	ST_TimeZoneInformation;
	MonthDays												:	WORD;
	LeapYear												:	BOOL;
	DayOfYear												:	WORD;
	WeekOfYear												:	WORD;
	UtcTimeFT												:	Tc2_Utilities.T_FILETIME; //Current UTC System/TwinCAT time T_FILETIME format, structure representing a 64-bit value with the a number of 100-nanosecond intervals since January 1, 1601 (UTC) (dwLowDateTime : DWORD / dwHighDateTime : DWORD)
	UtcTimeSTRUCT											:	Tc2_Utilities.TIMESTRUCT; //Current UTC System/TwinCAT time in TIMESTRUCT format
	UtcTimezoneBias											:	DINT;   //Total timezone bias in minutes to UTC 
	TimeDT													:	DATE_AND_TIME;	//Current time in DATE_AND_TIME format: DT#1970-01-01-00:00 -> DT#2106-02-06-06:28:15
	TimeTOD													:	TOD; //Current time in TOD format, range from TOD#00:00 -> TOD#1193:02:47.295
	TimeFT													:	Tc2_Utilities.T_FILETIME; //Current time in T_FILETIME format, structur representing a 64-bit value with the a number of 100-nanosecond intervals since January 1, 1601 (UTC) (dwLowDateTime : DWORD / dwHighDateTime : DWORD)
	TimeSTRUCT												:	Tc2_Utilities.TIMESTRUCT; //Current time in TIMESTRUCT format
	Datestamp												:	DATE; //D#1970-01-01 -> D#2106-02-06
	DateStr													:	STRING(15);	(* dd.mm.jj or mm.dd.jj *)	
	TimeStr													:	STRING(15);	(* hh:mm:ss.xxx or hh:mm:ss.xxxPM/AM *)
	TimeStamp												:	STRING(25); (* DateStr + TimeStr *)	
	TimeStamp2												:	STRING(25); (* YYYY-MM-DDTHHMMSS for example YYYY-MM-DD_HHMMSS_Name.txt *)
	TimeStamp3												:	STRING(25); (* YYYY-MM-DD-hh:mm:ss.xxx *)
	DateStrISO												:	STRING(15);	(* jj-mm-dd *)
	TimeStrISO												:	STRING(15);	(* hh:mm:ss *)
	TimeStampISO											:	STRING(25);	(* jj-mm-dd'T'hh:mm:ss.xxms *)	
	TimeStampStartup										:	DATE_AND_TIME; //Timestamp of startup
	DCTime													:	Tc2_EtherCAT.T_DCTIME64; //Current TwinCAT distributed clock time in 64-bit T_DCTIME64 format. The smallest unit is a nanosecond.
	DCTimeSTRUCT											:	Tc2_Utilities.TIMESTRUCT;//Current TwinCAT distributed clock time in TIMESTRUCT format
END_VAR
VAR
	(* Inst. Get Taskindex *)
	InstGETCURTASKINDEX										: 	GETCURTASKINDEX;
	InstLocalSystemTime										:	FB_LocalSystemTime;
	InstGetSystemTime										:	GetSystemTime;
	InstNtSetLocalTime										:	NT_SetLocalTime := (NETID := '', TMOUT := DEFAULT_ADS_TIMEOUT);
	InstTimeZoneInfo										:	FB_GetTimeZoneInformation;
	InstCpuCouter											:	GETCPUCOUNTER;
	InstGetDevIdent											:	FB_GetDeviceIdentificationEx;
	_OnlineChangeCount										: 	UDINT; 
	_sec													:	WORD;
	_hour													:	WORD;
	_Init													:	BOOL;
END_VAR

	(* Evaluate the PlcAppSystemInfo and and get sytstem timestamp					*)
	(********************************************************************************)
	
(* Get Current Task Index ************************************************************************)
	IF InstGETCURTASKINDEX.index = 0 then InstGETCURTASKINDEX(index => TaskIndex); END_IF

(* Read System Info Current Task *****************************************************************)	
	(* Get static information and boot error messages *)
	IF TwinCAT_SystemInfoVarList._TaskInfo[InstGETCURTASKINDEX.Index].FirstCycle 
	THEN
		AppTimestampDT										:= TwinCAT_SystemInfoVarList._AppInfo.AppTimestamp;
		AppTimestamp										:= DT_TO_STRING(AppTimestampDT);
		AppTimestamp										:= DELETE(AppTimestamp,3,1);
			
		TaskIndex											:= InstGETCURTASKINDEX.Index;
		TaskCnt 											:= TwinCAT_SystemInfoVarList._AppInfo.TaskCnt;
		
		ObjId												:= TwinCAT_SystemInfoVarList._AppInfo.ObjId;
		AppName												:= TwinCAT_SystemInfoVarList._AppInfo.AppName;	
		ProjectName											:= TwinCAT_SystemInfoVarList._AppInfo.ProjectName;	
		AdsPort												:= TwinCAT_SystemInfoVarList._AppInfo.AdsPort;	
			
		Flags												:= TwinCAT_SystemInfoVarList._AppInfo.Flags;
//		PersistentStatus									:= TwinCAT_SystemInfoVarList._AppInfo.PersistentStatus;
		
		BootDataLoaded										:= TwinCAT_SystemInfoVarList._AppInfo.BootDataLoaded;
		OldBootData											:= TwinCAT_SystemInfoVarList._AppInfo.OldBootData;
		NoBootDataLoaded									:= NOT BootDataLoaded AND NOT OldBootData;
		BSODOccured 										:= TwinCAT_SystemInfoVarList._AppInfo.BSODOccured;
		
		CycleTime         									:= TwinCAT_SystemInfoVarList._TaskInfo[TaskIndex].CycleTime;
		CycleTimeNS         								:= TwinCAT_SystemInfoVarList._TaskInfo[TaskIndex].CycleTime * 100;
		CycleTimeT											:= LREAL_TO_TIME(UDINT_TO_LREAL(CycleTime) * 0.0001 );
		CycleTimeLT											:= TO_LTIME(CycleTimeNS);	
		CycleTimeFloat										:= (UDINT_TO_LREAL(CycleTime) * 0.0001 / 1000.0);	
		
	ELSIF ResetTrig
	THEN
		resetBootInfo();
	ELSIF NOT Enable
	THEN
		RETURN;
	END_IF
	
	OnlineChangeCount										:= TwinCAT_SystemInfoVarList._AppInfo.OnlineChangeCnt;
	OnlineChange											:= _OnlineChangeCount <> OnlineChangeCount;
	_OnlineChangeCount										:= OnlineChangeCount;
	LoggedIn 												:= TwinCAT_SystemInfoVarList._AppInfo.LoggedIn;
	ShutdownInProgress 										:= TwinCAT_SystemInfoVarList._AppInfo.ShutdownInProgress;
	LicensesPending 										:= TwinCAT_SystemInfoVarList._AppInfo.LicensesPending;
	TComSrvPtr												:= TwinCAT_SystemInfoVarList._AppInfo.TComSrvPtr;
	TwinCAT_SystemInfoVarList._AppInfo.KeepOutputsOnBP		:= KeepOutputsOnBP;		

(* CPU System counter ****************************************************************************)
	InstCpuCouter(cpuCntLoDW => CpuCounter);	
	MEMCPY(ADR(CpuCounter) + SIZEOF(InstCpuCouter.cpuCntHiDW),ADR(InstCpuCouter.cpuCntHiDW),SIZEOF(InstCpuCouter.cpuCntHiDW));
	
(* Get device identification structure ***********************************************************)
	InstGetDevIdent(
		bExecute	:= NOT Options.3, 
		tTimeout	:= , 
		sNetId		:= , 
		bBusy		=> , 
		bError		=> , 
		nErrorID	=> , 
		stDevIdent	=> );	
	pDevIdent												:= ADR(InstGetDevIdent.stDevIdent);
	IF NOT InstGetDevIdent.bBusy
	THEN
		DevIdentValid										:= NOT InstGetDevIdent.bError;
		
		IF InstGetDevIdent.bError AND ResetTrig
		THEN
			InstGetDevIdent(bExecute := FALSE);			
		END_IF
	ELSE	
		DevIdentValid										:= FALSE;
	END_IF
	
(* Read timezone information for one time ******************************************************)
	IF Enable AND NOT InstTimeZoneInfo.bExecute
		OR InstTimeZoneInfo.bBusy
	THEN
		InstTimeZoneInfo(
			sNetID	:= , 
			bExecute:= TRUE, 
			tTimeout:= , 
			bBusy	=> , 
			bError	=> , 
			nErrID	=> , 
			tzID	=> TimeZoneId, 
			tzInfo	=> TimeZoneInfo);
		IF NOT InstTimeZoneInfo.bBusy AND NOT InstTimeZoneInfo.bError
		THEN
			UtcTimezoneBias									:= -1 * (TimeZoneInfo.bias + TimeZoneInfo.daylightBias);
		ELSE
			UtcTimezoneBias									:= 0;
		END_IF
	ELSIF NOT Enable AND InstTimeZoneInfo.bExecute	
	THEN
		InstTimeZoneInfo(bExecute:= FALSE);
	END_IF
		
(* Actual time in DCTIME format ****************************************************************)
	DCTime													:= F_GetActualDcTime64();
	DCTimeSTRUCT											:= DCTIME64_TO_SYSTEMTIME(DCTime);

(* Get TwinCAT/system time in UTC Filetime format ******************************************************)
	InstGetSystemTime(
		 timeLoDW=>UTCTimeFT.dwLowDateTime,
		 timeHiDW=>UTCTimeFT.dwHighDateTime);
		 
	UTCTimeSTRUCT											:= FILETIME_TO_SYSTEMTIME(UTCTimeFT);	 
		
(* evalutate systemtime ************************************************************************)
	InstLocalSystemTime(
		sNetID		:= '',
		bEnable		:= Enable,
		dwCycle		:= SEL(InstNtSetLocalTime.START, RtcSyncCylce, 1), //Short update cylce to read windows time after it was set
		dwopt		:= (* Default *),
		tTimeout	:= (* Default *),
		bValid		=> ,
		systemTime	=> TimeSTRUCT,
		tzID		=> );
				
	IF InstLocalSystemTime.bValid 
	THEN				
		//Update cyclic
		TimeFT												:= SYSTEMTIME_TO_FILETIME(TimeSTRUCT);
		TimeDT 												:= SYSTEMTIME_TO_DT(TimeSTRUCT);
		TimeStamp3											:= SYSTEMTIME_TO_STRING(TimeSTRUCT);
		TimeTOD												:= SEL(Options.2 ,TO_TOD(TimeDT)  , DWORD_TO_TOD(TO_DWORD(TO_TOD(TimeDT)) + TimeSTRUCT.wMilliseconds));  
		TimeStrISO											:= DELETE(TO_STRING(TimeTOD),4,1);
		TimeStampISO										:= CONCAT(DateStrISO , CONCAT('T',TimeStrISO));	
			
		//Create time format
		IF Options.1
		THEN (* US time format hh.mm.ss AM/PM ***************)
			IF TimeSTRUCT.wHour < 10 
			THEN
				TimeStr 									:= CONCAT('0',WORD_TO_STRING(TimeSTRUCT.wHour));
			ELSIF TimeSTRUCT.wHour > 12 
			THEN
				TimeStr 									:= WORD_TO_STRING(TimeSTRUCT.wHour - 12);
				IF TimeSTRUCT.wHour - 12 < 10
				THEN
					TimeStr									:= CONCAT('0',TimeStr);
				END_IF
			ELSE         									
				TimeStr 									:= WORD_TO_STRING(TimeSTRUCT.wHour);
			END_IF		                                    
		ELSE  (* Time hh.mm.ss.xxms ***************)          
			IF TimeSTRUCT.wHour < 10                        
			THEN                                            
				TimeStr 									:= CONCAT('0',WORD_TO_STRING(TimeSTRUCT.wHour));
			ELSE        									
				TimeStr 									:= WORD_TO_STRING(TimeSTRUCT.wHour);
			END_IF			
		END_IF
		
		TimeStr 											:= CONCAT(TimeStr,':');
		
		IF TimeSTRUCT.wMinute < 10 
		THEN
			TimeStr 										:= CONCAT(TimeStr,CONCAT('0',WORD_TO_STRING(TimeSTRUCT.wMinute)));
		ELSE
			TimeStr 										:= CONCAT(TimeStr,WORD_TO_STRING(TimeSTRUCT.wMinute));
		END_IF
		
		TimeStr 											:= CONCAT(TimeStr,':');
		
		IF TimeSTRUCT.wSecond < 10 
		THEN
			TimeStr 										:= CONCAT(TimeStr,CONCAT('0',WORD_TO_STRING(TimeSTRUCT.wSecond)));
		ELSE        										
			TimeStr 										:= CONCAT(TimeStr,WORD_TO_STRING(TimeSTRUCT.wSecond));
		END_IF  
												
		IF Options.2
		THEN //add ms to timestamp
			TimeStr 										:= CONCAT(TimeStr,'.');
			TimeStr 										:= CONCAT(TimeStr,WORD_TO_STRING(TimeSTRUCT.wMilliseconds));
		END_IF
		
		IF Options.1
		THEN //US time format
			TimeStr 										:= CONCAT(TimeStr,SEL(TimeSTRUCT.wHour > 12,' AM', ' PM'));
		END_IF
		
		(* TimeStamp Format DE: DD.MM.YY-Stunde:Minute:Sekunde.xxx,*)
		TimeStamp 											:= CONCAT(DateStr,'-');
		TimeStamp 											:= CONCAT(TimeStamp,TimeStr);
		
		IF _hour <> TimeSTRUCT.wHour OR NOT _Init
		THEN
			_Hour											:= TimeSTRUCT.wHour;		
			//Create date in US fromat with seperator / ************************************************
			IF Options.0
			THEN (* Date mm/dd/jj ********************)
				IF TimeSTRUCT.wMonth < 10 
				THEN
					DateStr 								:= CONCAT('0',WORD_TO_STRING(TimeSTRUCT.wMonth));
				ELSE        								
					DateStr 								:= WORD_TO_STRING(TimeSTRUCT.wMonth);
				END_IF		                                
				DateStr 									:= CONCAT(DateStr,DateStrSeperator);
				IF TimeSTRUCT.wDay < 10                     
				THEN                                        
					DateStr 								:= CONCAT(DateStr,CONCAT('0',WORD_TO_STRING(TimeSTRUCT.wDay)));
				ELSE        								
					DateStr 								:= CONCAT(DateStr,WORD_TO_STRING(TimeSTRUCT.wDay));
				END_IF                                      
															
				DateStr 									:= CONCAT(DateStr,DateStrSeperator);
				DateStr 									:= CONCAT(DateStr,RIGHT(WORD_TO_STRING(TimeSTRUCT.wYear),2));		
		                                                    
			ELSE (* Date dd.mm.jj ********************)	    
				IF TimeSTRUCT.wDay < 10                     
				THEN                                        
					DateStr 								:= CONCAT('0',WORD_TO_STRING(TimeSTRUCT.wDay));
				ELSE        								
					DateStr 								:= WORD_TO_STRING(TimeSTRUCT.wDay);
				END_IF                                      
				DateStr 									:= CONCAT(DateStr,DateStrSeperator);
				IF TimeSTRUCT.wMonth < 10                   
				THEN                                        
					DateStr 								:= CONCAT(DateStr,CONCAT('0',WORD_TO_STRING(TimeSTRUCT.wMonth)));
				ELSE        								
					DateStr 								:= CONCAT(DateStr,WORD_TO_STRING(TimeSTRUCT.wMonth));
				END_IF                                      
															
				DateStr 									:= CONCAT(DateStr,DateStrSeperator);
				DateStr 									:= CONCAT(DateStr,RIGHT(WORD_TO_STRING(TimeSTRUCT.wYear),2));	
			END_IF      

			DateStrISO										:= DELETE(TO_STRING(TO_DATE(TimeDT)),2,1);
			
			(* information of year *)                       
			MonthDays										:= F_GetMaxMonthDays(TimeSTRUCT.wYear,TimeSTRUCT.wMonth);
			LeapYear										:= F_YearIsLeapYear(TimeSTRUCT.wYear) ;
			WeekOfYear										:= F_GetWeekOfTheYear(TimeDT);
			DayOfYear										:= F_GetDOYOfYearMonthDay(TimeSTRUCT.wYear,TimeSTRUCT.wMonth,TimeSTRUCT.wDay);
			DateStamp										:= TO_DATE(TimeDT);		
             
			IF NOT _Init 
			THEN	
				_INIT										:= TRUE; 
				TimeStampStartup							:= SYSTEMTIME_TO_DT(TimeSTRUCT);
			END_IF
                       
		END_IF //hour
		
		IF _sec <> TimeSTRUCT.wSecond 
		THEN	
			_sec 											:= TimeSTRUCT.wSecond;
														
			(* TimeStamp2 FileName YYYY-MM-DD_HHMMSS *)
			TimeStamp2										:= CONCAT(DateStrISO , '_');
			IF TimeSTRUCT.wHour < 10                    	
			THEN                                        	
				TimeStamp2 									:= CONCAT(TimeStamp2,CONCAT('0',WORD_TO_STRING(TimeSTRUCT.wHour)));
			ELSE           									
				TimeStamp2 									:= CONCAT(TimeStamp2,WORD_TO_STRING(TimeSTRUCT.wHour));
			END_IF                                      	
			IF TimeSTRUCT.wMinute < 10                  	
			THEN                                        	
				TimeStamp2 									:= CONCAT(TimeStamp2,CONCAT('0',WORD_TO_STRING(TimeSTRUCT.wMinute)));
			ELSE           									
				TimeStamp2 									:= CONCAT(TimeStamp2,WORD_TO_STRING(TimeSTRUCT.wMinute));
			END_IF                                      	
			IF TimeSTRUCT.wSecond < 10                  	
			THEN                                        	
				TimeStamp2 									:= CONCAT(TimeStamp2,CONCAT('0',WORD_TO_STRING(TimeSTRUCT.wSecond)));
			ELSE           									
				TimeStamp2 									:= CONCAT(TimeStamp2,WORD_TO_STRING(TimeSTRUCT.wSecond));
			END_IF
		END_IF //second update
														
	END_IF

(* set system time *****************************************************************************)
	InstNtSetLocalTime(
		NETID		:= , 
		TIMESTR		:= , 
		START		:= , // Start by Methode "SetSysTime" 
		TMOUT		:= , 
		BUSY		=> , 
		ERR			=> ); 
	
	IF InstNtSetLocalTime.START AND NOT InstNtSetLocalTime.BUSY
	THEN //Take care that all timestamp get updated after set a new time
		InstNtSetLocalTime.START							:= FALSE;	
		_Init												:= FALSE;								
	END_IF
	
(**************************************************************************************************)

PROPERTY PUBLIC optAddmsToTimeString : BOOL
GET
optAddmsToTimeString := Options.2;
END_GET
SET
Options.2 := optAddmsToTimeString;
END_SET
END_PROPERTY

PROPERTY PUBLIC  optDisableReadDeviceIdentification : BOOL
GET
optDisableReadDeviceIdentification := Options.3;
END_GET
SET
Options.3 := optDisableReadDeviceIdentification;
END_SET
END_PROPERTY

PROPERTY PUBLIC optEnableUSDateFormat : BOOL
GET
optEnableUSDateFormat := Options.0;
END_GET
SET
Options.0 := optEnableUSDateFormat;
END_SET
END_PROPERTY

PROPERTY PUBLIC optEnableUSTimeFormat : BOOL
GET
optEnableUSTimeFormat := Options.1;
END_GET
SET
Options.1 := optEnableUSTimeFormat;
END_SET
END_PROPERTY

METHOD PUBLIC resetBootInfo : BOOL  //Return value = TRUE if execution finished
VAR_INPUT
END_VAR
OldBootData 												:= FALSE;
BSODOccured													:= FALSE;
NoBootDataLoaded											:= FALSE;
resetBootInfo												:= TRUE;
END_METHOD

METHOD PUBLIC setSysTime  : BOOL //Return value = TRUE if execution finished
VAR_INPUT
	TimeStruct		: TIMESTRUCT;
END_VAR
InstNtSetLocalTime(
		NETID		:= '', 
		TIMESTR		:= TimeStruct, 
		START		:= NOT InstNtSetLocalTime.START AND TimeStruct.wYear > 2000 
						AND TimeStruct.wDay > 0 AND TimeStruct.wMonth	< 32	
						AND TimeStruct.wMonth > 0 AND TimeStruct.wMonth	< 13	
						AND TimeStruct.wHour >= 0 AND TimeStruct.wHour	< 24	
						AND TimeStruct.wMinute >= 0 AND TimeStruct.wMinute < 60
						AND TimeStruct.wSecond >= 0 AND TimeStruct.wSecond < 60				
						OR InstNtSetLocalTime.BUSY, 
		TMOUT		:= , 
		BUSY		=> , 
		ERR			=> , 
		ERRID		=> );
		
setSysTime													:= InstNtSetLocalTime.BUSY;
END_METHOD

END_FUNCTION_BLOCK

// POUs/Fieldbus/EtherCAT/EcDiagBase
{attribute 'no_check'}
FUNCTION_BLOCK EcDiagBase
VAR_OUTPUT CONSTANT         								
	MIN_SLAVES												: 	UINT := 1;
	MAX_SLAVES												: 	UINT := PARAM.ETHERCAT_DIAG_MAX_SLAVES;	//EC_MAX_SLAVES = 65535 Slaves;
END_VAR
VAR_INPUT
	Enable													:	BOOL := TRUE;//FB will be processed as long as enable is TRUE 
	
	DelReadSlavesDiag										:	TIME := T#2S; //Damping time to read diagnostic if error is detected 
	SourceId												: 	UDINT := 103000; //Multisource id 
(* Components *)            								
	IO														:	EcMasterIO;
END_VAR                     								
VAR_OUTPUT                  								
	MasterOK												:	BOOL; 	//TRUE when Master/EtherCAT is OK
	SlavesOK												:	BOOL;	//TRUE if no slave is in error state
	NoOfSlavesNOK											:	UINT;
	NoOfMissedSlaves										:	INT; //No of slaves missed incl. hot connect slaves 
	NoOfHotConnectGroups									:	UINT;
	NoOfHotConnectSlaves									:	UINT;
	
	pSlaveInfoData											:	POINTER TO ARRAY [MIN_SLAVES..MAX_SLAVES] OF EC_SLAVE_DIAG_INFO_DATA := ADR(SlavesDiag.InfoData); //configures slaves			
	DiagBusy												:	BOOL;
	ErrorReadDiag											:	BOOL;
END_VAR
VAR
(* Local  ***********************************************************)
	MemSlaveCount											:	UINT;
	MemDevState												:	UINT;
	InitDone												:	BOOL;
	
(* trigger ********************************************************)
	rtReadDiag												: r_Trig;

(* Timer **********************************************************)
	tonDelTrigDiag											:	ton;

(* events *********************************************************)

(* function-block *************************************************)
	SlavesDiag												:	EcSlavesDiag;
	
(* dummy **********************************************************)
	idx,i													:	INT;											
END_VAR

(* Base diagnostic of EtherCAT 					*)
(************************************************)

(* Work IO *************************************************)
	IO();

(* trigger slaves diag *************************************************************)
	IF NOT tonDelTrigDiag.IN AND NOT SlavesDiag.Busy
		AND( 
		IO.FramesWcStateChanged
		OR MemDevState <> IO.DevState
		OR MemSlaveCount <> IO.SlaveCountTotal
		OR NOT InitDone)
	THEN
		tonDelTrigDiag(IN := TRUE , PT := DelReadSlavesDiag);
	END_IF
	//Run delay	
	tonDelTrigDiag();
	
	rtReadDiag(CLK := Enable AND tonDelTrigDiag.Q);
	IF rtReadDiag.Q 
	THEN 	
		tonDelTrigDiag(IN := FALSE); //Restart timer
		SlavesDiag.optReadScannedSlaves						:= MemSlaveCount <> IO.SlaveCountTotal OR NoOfMissedSlaves > 0 OR SlavesDiag.InvalidVPRS; //Scan slaves if invalid VPRS or HC groups are configured
	//	SlavesDiag.optSortInfoData 							:= ;
	//	SlavesDiag.optUpdateTopoData						:= ;
	//	SlavesDiag.optUpdateConfigData 						:= ;
		
	 	MemSlaveCount 										:= IO.SlaveCountTotal;
		MemDevState 										:= IO.DevState;
		InitDone											:= TRUE;
	END_IF
	SlavesDiag(Execute := rtReadDiag.Q,MasterAmsNetId := IO.AmsNetIdStr, NoOfSlavesNOK => NoOfSlavesNOK, NoOfHCGroups => NoOfHotConnectGroups, NoOfHCSlaves => NoOfHotConnectSlaves, Busy => DiagBusy , Error => ErrorReadDiag);		
	pSlaveInfoData											:= ADR(SlavesDiag.InfoData);
		
(***********************************************************************************)
	MasterOK 												:= IO.DevStateBits.NoError;
	SlavesOK												:= MasterOK AND SlavesDiag.NoOfSlavesNOK = 0;
	NoOfMissedSlaves										:= TO_INT(IO.CfgSlaveCount) - TO_INT(IO.SlaveCountTotal);
	
(*********************************************************************************)

END_FUNCTION_BLOCK

// POUs/Fieldbus/EtherCAT/EcDiagBase_wEvents
{attribute 'no_check'}
FUNCTION_BLOCK EcDiagBase_wEvents EXTENDS EcDiagBase
VAR_OUTPUT CONSTANT         								
END_VAR
VAR_INPUT
	ConfirmTrig												:	BOOL;
END_VAR                     								
VAR_OUTPUT                  								
	{attribute 'displaymode':='binary'}
	EventStatus												:	DWORD;
END_VAR
VAR
(* Local  ***********************************************************)

	
(* trigger ********************************************************)


(* Timer **********************************************************)


(* events *********************************************************)
	Event													:	EventHandlingGrp10;
	
(* function-block *************************************************)

	
(* dummy **********************************************************)
										
END_VAR

(* Base diagnostic of EtherCAT with events		*)
(************************************************)

(* Call super  *************************************************)
	SUPER^();
	
(* Fire events **********************************************************************)
	_callEvents();
	
(**************************************************************************************)

METHOD PRIVATE _callEvents : BOOL
VAR_INPUT
END_VAR
(* Events anzeigen ***************************************************)
	(* Init events *)
	IF Event.no[1].Text1 <> IO.Name
	THEN
		FOR i := Event.MIN_EVENT TO Event.MAX_EVENT 
		DO
			Event.no[i].Text1								:= IO.Name;
		END_FOR
	END_IF 

	(* Master Error Event *)
	
	Event.no[1].Flag										:= NOT IO.DevStateBits.NoError AND NOT IO.DevStateChanged AND NOT ConfirmTrig;
	Event.no[1].pText3										:= ADR(IO.DevStateText);

	(* Error Port Link *)
	Event.no[2].Flag										:=(NOT IO.LinkOK_PortA OR NOT IO.LinkOK_PortB) AND NOT SlavesDiag.Busy AND NOT tonDelTrigDiag.IN;
	IF Event.no[2].Flag
	THEN
		Event.no[2].Text2									:= TO_STRING(NoOfMissedSlaves);
		Event.no[2].pText3									:= ADR(SlavesDiag.FirstErrorSlave.ConfigName);	
	END_IF

	(* No Slave Com *)
	Event.no[3].Flag										:= IO.AllFramesMissing AND NoOfMissedSlaves = 0 AND NOT IO.DevStateChanged AND NOT SlavesDiag.Busy AND NOT tonDelTrigDiag.IN;
	IF Event.no[3].Flag
	THEN
		Event.no[3].Text2									:= CONCAT(CONCAT('(',SlavesDiag.FirstErrorSlave.ConfigType), CONCAT(') , ',TO_STRING(NoOfMissedSlaves))) ;
		Event.no[3].pText3									:= ADR(SlavesDiag.FirstErrorSlave.ConfigName);	
	END_IF

	(* Slave State Error *)
	Event.no[4].Flag										:= NoOfSlavesNOK > 0 AND NOT IO.DevStateChanged AND NOT SlavesDiag.Busy AND NOT tonDelTrigDiag.IN;
	IF Event.no[4].Flag
	THEN
		Event.no[4].Text2									:= CONCAT(SlavesDiag.FirstErrorSlave.DevStateText , CONCAT(', Name: ', SlavesDiag.FirstErrorSlave.ConfigName));
		Event.no[4].pText3									:= ADR(SlavesDiag.FirstErrorSlave.ConfigTypeIdentity);	
	END_IF
	
	(* Slave Count Error *)
	Event.no[5].Flag										:= NoOfMissedSlaves <> 0 AND NoOfSlavesNOK > 0 AND NOT ConfirmTrig AND NOT SlavesDiag.Busy AND NOT tonDelTrigDiag.IN;
	IF Event.no[5].Flag
	THEN
		Event.no[5].Text2									:= CONCAT('Cfg Slaves:',CONCAT(TO_STRING(IO.CfgSlaveCount),CONCAT(' | Found:',TO_STRING(IO.SlaveCountTotal))));
		Event.no[5].pText3									:= ADR(SlavesDiag.FirstErrorSlave.ConfigName);
	END_IF	
		
	(* Frm Wc Error  *)
	Event.no[6].Flag										:= FALSE ;          									
	IF Event.no[6].Flag 									
	THEN    
		Event.no[6].Text2									:= '';            									
		Event.no[6].pText3									:= ADR(IO.DevStateText);
	END_IF	
	
	(* Watchdog triggered  *)
	Event.no[7].Flag										:= io.DevStateBits.WatchdogTriggered;	
	IF Event.no[7].Flag 
	THEN 
		Event.no[7].pText3									:= ADR(IO.DevStateText);
	END_IF	
	
	(* DC not in sync  *)
	Event.no[8].Flag										:= IO.DevStateBits.DcNotInSync;
	IF Event.no[8].Flag 
	THEN 
		Event.no[8].pText3									:= ADR(IO.DevStateText);
	END_IF	
	
	(* Out of send ressources  *)
	Event.no[9].Flag										:= IO.DevStateBits.OutOfSendResources;
	IF Event.no[9].Flag 
	THEN 
		Event.no[9].pText3									:= ADR(IO.DevStateText);
	END_IF	

	(* IO locked  *)
	Event.no[10].Flag										:= IO.DevStateBits.IOLockedAfterLinkError;		
	IF Event.no[10].Flag 
	THEN 
		Event.no[10].pText3									:= ADR(IO.DevStateText);
	END_IF
	
	(* Work EventCtrl *)
	Event(
		ConfirmTrig	:= ConfirmTrig,
		SourceId	:= SourceId ,
		no			:= ,
		Disable		:= NOT Enable,
		AutoConfirm := ,
		Status		=> EventStatus);
		
(*****************************************************************************)
END_METHOD

METHOD PUBLIC confirm : bool
VAR_INPUT
END_VAR
confirm			:= Event.confirm();
END_METHOD

END_FUNCTION_BLOCK

// POUs/Fieldbus/Profibus/ProfibusMasterDiag
{attribute 'no_check'}
FUNCTION_BLOCK ProfibusMasterDiag
VAR_INPUT                               					
	Enable													:	BOOL := FALSE;		//FB will be processed as long as enable is TRUE 	
	ResetTrig													:	BOOL := FALSE;		//Resets error with rising edge 
	SourceId												:	UDINT := 103020; 	//default
END_VAR                                 	
VAR_OUTPUT                              	
	IO														:	ProfiBusMasterIO;
END_VAR
VAR
(* trigger ********************************************************)
		
(* events *********************************************************)
	EventMasterError										:	EventHandling;
	EventNoteError											:	ARRAY[1..PARAM.PROFIBUS_MASTER_DEV_IO_MAX_SLAVES] OF EventHandling;
(* function-block *************************************************)
	
(* dummy **********************************************************)	
	i														:	INT;
END_VAR

	(* ProfiBus master diagnosis for EL6731 and slaves	V2.0	*)
	(************************************************************)

(* Work IO ***********************************************)
	IO();

(* Master error ******************************************************)
	EventMasterError(
		Flag			:= IO.Error <> 0 AND Enable,
		ConfirmTrig		:= ResetTrig OR NOT Enable,
		MsgId			:= 1,
		SourceId		:= SourceId,
		Class			:= ,
		Text1			:= ,
		Text2			:= USINT_TO_STRING(IO.Error),
		pText3			:= ADR(IO.Name),
		State			=> );
		
(* Slave note error **************************************)
	FOR i := IO.MIN_SLAVES TO IO.MAX_SLAVES DO		
		EventNoteError[i](
			Flag		:= IO.SlaveDpStates[i] <> 0 AND Enable,
			ConfirmTrig := ResetTrig OR NOT Enable,
			MsgId		:= TO_UINT(i + 1),
			Text1		:= TO_STRING(i),
			Text2		:= TO_STRING(IO.SlaveDpStates[i]),
			pText3		:= ADR(IO.Name),
			SourceId	:= );
		
 	END_FOR
	

		
(*********************************************************)

END_FUNCTION_BLOCK

// POUs/Fieldbus/Profibus/ProfibusMasterIO
{attribute 'no_check'}
//EL6731 Profibus Master IOs via EtherCAT
FUNCTION_BLOCK ProfibusMasterIO
VAR_OUTPUT CONSTANT
	MIN_SLAVES												:	INT := 1;
	MAX_SLAVES												:	INT := PARAM.PROFIBUS_MASTER_DEV_IO_MAX_SLAVES;
END_VAR
VAR_INPUT
END_VAR
VAR_OUTPUT
	DevId											AT %I*	: 	UINT; 		//Map to Device Id or EtherCAT Master DevId
	AdsAddr											AT %I*	:	AMSADDR;	//Structure of AdsAddr
	AmsNetIdStr												:	T_AmsNetId;	//shows string of AmsNetId 
	Error											AT %I*	:	USINT;		//No of Slaves with an state <> 0
	ActualModulo		 							AT %I*	:	USINT;		
	DiagFlag										AT %I*	:	BOOL;		//TRUE when diagnostic values are available
	Name													:	STRING(30);
                            					             	
	SlaveDpStates									AT %I*	:	ARRAY[MIN_SLAVES..MAX_SLAVES] OF USINT;
	SlaveExtDiagFlags								AT %I*	:	ARRAY[MIN_SLAVES..MAX_SLAVES] OF BOOL;
END_VAR                     					             	
VAR                         	                             	
	IOF_GetBoxNameByAddr									:	IOF_GetBoxNameByAddr := (NETID := '', TMOUT := DEFAULT_ADS_TIMEOUT);
END_VAR

(* Profibus Master IO diag										      	 		*)
(********************************************************************************)

(* Get name ******************************************************************************)
IF Name = ''
	AND AdsAddr.port <> 0 AND DevId <> 0
	OR IOF_GetBoxNameByAddr.BUSY
	OR IOF_GetBoxNameByAddr.START
THEN
	AmsNetIdStr												:= F_CreateAmsNetId(nIds := AdsAddr.netId);

	IF AmsNetIdStr = '0.0.0.0.0.0' THEN
		AmsNetIdStr	:= '';
	END_IF
		
	IOF_GetBoxNameByAddr(
		NETID		:= AmsNetIdStr , 
		DEVICEID	:= UINT_TO_UDINT(DevId) ,
		BOXADDR		:= AdsAddr.port ,
		START		:= Name = '' AND NOT IOF_GetBoxNameByAddr.BUSY,
		TMOUT		:= ,
		BOXNAME		=> name);
END_IF
(********************************************************************************)

END_FUNCTION_BLOCK

// POUs/Fieldbus/Profinet/ProfiNetMasterDiag
{attribute 'no_check'}
FUNCTION_BLOCK ProfiNetMasterDiag
VAR_INPUT                               					
	Enable													:	BOOL := FALSE;
	ResetTrig												:	BOOL := FALSE;
	SourceId												:	UDINT := 103040; (* default *)
END_VAR                                 	
VAR_OUTPUT                              	
	IO														:	ProfiNetMasterIO;
END_VAR
VAR
(* trigger ********************************************************)
	
(* events *********************************************************)
	EventMasterError										:	EventHandling;
	EventBoxError											:	ARRAY[1..PARAM.PROFINET_MASTER_DEV_IO_MAX_BOX] OF EventHandling;
	
(* function-block *************************************************)
	
(* dummy **********************************************************)	
	i														:	INT;
END_VAR

	(* ProfiNET master diagnosis for EL6631	and boxes	V2.0	*)
	(************************************************************)

(* Work IO ***********************************************)
	IO();
	
(* Master error *******************************************)
	EventMasterError(
		Flag				:= IO.PnIoError <> 0 AND Enable,
		ConfirmTrig			:= ResetTrig OR NOT Enable,
		MsgId				:= 1,
		SourceId			:= SourceId,
		Class				:= ,
		Text1				:= TO_STRING(IO.PnIoError),
		Text2				:= ,
		pText3				:= ADR(IO.Name),
		State				=> );

(* Box error *********************************************)
	FOR i := IO.MIN_BOX TO IO.MAX_BOX DO
		EventBoxError[i](
			Flag			:= IO.PnIoBoxDiags[i] <> 0 AND Enable,
			ConfirmTrig		:= ResetTrig OR NOT Enable,
			MsgId			:= TO_UINT(i + 1),
			SourceId		:= SourceId,
			Class			:= ,
			Text1			:= TO_STRING(IO.PnIoBoxDiags[i]),
			Text2			:= TO_STRING(i),
			pText3			:= ADR(IO.Name),
			State			=> );
 	END_FOR

(*********************************************************)

END_FUNCTION_BLOCK

// POUs/Fieldbus/Profinet/ProfiNetMasterIO
{attribute 'no_check'}
//EL6731 Profibus Master IOs via EtherCAT
FUNCTION_BLOCK ProfiNetMasterIO
VAR_OUTPUT CONSTANT
	MIN_BOX												:	INT := 1;
	MAX_BOX												:	INT := PARAM.PROFINET_MASTER_DEV_IO_MAX_BOX;
END_VAR
VAR_INPUT
	DevCtrl			 								AT %Q*	:	UINT;
	PnIoBoxCtrl										AT %Q*	:	ARRAY[MIN_BOX ..MAX_BOX] OF UINT;
END_VAR
VAR_OUTPUT
//EL Parameter
	AdsAddr											AT %I*	:	AMSADDR; //Link to device Ads addesss
	DevID											AT %I*	:	UINT;		//Device or EtherCAT master device id
	AmsNetIdStr												:	T_AmsNetId; //Device AMS address as string
	
//Device parameter
	DevState		 								AT %I*	:	UINT;		//Link to master device state
	PnIoError										AT %I*	:	UINT;		//Link to master IO error 
	PnIoDiag										AT %I*	:	UINT;		//Link to master IO diag 
   	Name													:	STRING(30);
                         				
//Box states	             	
	PnIoBoxStates									AT %I*	:	ARRAY[MIN_BOX ..MAX_BOX] OF UINT; //Link to box state
	PnIoBoxDiags									AT %I*	:	ARRAY[MIN_BOX ..MAX_BOX] OF UINT; //Link to box diag	
END_VAR                     					             	
VAR       
	IOF_GetBoxNameByAddr									:	IOF_GetBoxNameByAddr;
END_VAR

(* Get Master Name *)
IF Name = ''
	AND AdsAddr.port <> 0
	OR IOF_GetBoxNameByAddr.BUSY
	OR IOF_GetBoxNameByAddr.START
THEN
	AmsNetIdStr												:= F_CreateAmsNetId(nIds := AdsAddr.netId);
		
	IF AmsNetIdStr = '0.0.0.0.0.0' THEN
		AmsNetIdStr	:= '';
	END_IF
	
	IOF_GetBoxNameByAddr(
		NETID			:= AmsNetIdStr, 
		DEVICEID		:= UINT_TO_UDINT(DevId) , 
		BOXADDR			:= AdsAddr.port,
		START			:= Name = '' AND NOT IOF_GetBoxNameByAddr.BUSY, 
		TMOUT			:= , 
		BUSY			=> , 
		ERR				=> , 
		ERRID			=> , 
		BOXNAME			=> name);

END_IF

END_FUNCTION_BLOCK

// POUs/FileHandling/Basic/FileHandling
{attribute 'no_check'}
//Wrapper for all file fucntions provided by lib Tc2_TcSystem.Lib, see Beckhoff information system for detailed information of each function. 
FUNCTION_BLOCK FileHandling EXTENDS FbBase
VAR_OUTPUT CONSTANT
	FNC_OPEN												:	INT := 0; //With this function a new file can be created, or a closed existing file can be re-opened for further processing
	FNC_READ												:	INT := 1; //With this function  the contents of an already opened file can be read. The file must have been already opened for read access
	FNC_WRITE												:	INT := 2; //Data can be written into a file with this function if it is opened in write mode
	FNC_PUTS												:	INT := 3; //The function writes strings to the file if it is opened in write mode
	FNC_GETS												:	INT := 4; //The function reads zero terminated strings from a file and moves the file pointer to the next line.(if pBuffer is <> 0, the read line will copied to the buffer as well)
	FNC_CLOSE												:	INT := 5; //With this function the file can be closed, and thereby placed into a defined state for further processing by other programs
	FNC_DELETE												:	INT := 6; //With this function the existing file can be deleted
	FNC_RENAME												:	INT := 7; //With this function the existing file can be renamed.
	FNC_REMOVEDIR											:	INT := 8; //This function removes a directory from the data medium. A directory containing data can not be removed!
	FNC_CREATEDIR											:	INT := 9; //This function creates new directories on the data medium.
	FNC_SEEK												:	INT := 10;//With this function the file pointer of an opened file can be set to a definable position
	FNC_TELL												:	INT := 11;//The function gets the current position of the file pointer. The position is expressed as an offset relative to the beginning of the stream.
	FNC_EOF													:	INT := 12;//The function tests for the end-of-file.
END_VAR             										                 										
VAR_INPUT           										
	Fnc														:	INT (FNC_OPEN..FNC_EOF) := FNC_OPEN; //Parameter for requested function
	AMSNetId												:	T_AmsNetId := ''; //Ams Net Id 
	Timeout													:	TIME := DEFAULT_ADS_TIMEOUT; //Ads timeout 
	Mode													:	DWORD := FOPEN_MODEAPPEND OR FOPEN_MODEPLUS OR FOPEN_MODETEXT; 
																			(* 	FOPEN_MODEREAD "r": Opens for reading. If the file does not exist or cannot be found, the call fails.
																				FOPEN_MODEWRITE  "w": Opens an empty file for writing. If the given file exists, its contents are destroyed.
																				FOPEN_MODEAPPEND  "a": Opens for writing at the end of the file (appending) without removing the EOF marker before writing new data to the file; creates the file first if it doesn’t exist.
																				FOPEN_MODEREAD OR FOPEN_MODEPLUS  "r+": Opens for reading and writing. The file must exist.
																				FOPEN_MODEWRITE OR FOPEN_MODEPLUS  "w+": Opens an empty file for both reading and writing. If the given file exists, its contents are destroyed.
																				FOPEN_MODEAPPEND OR FOPEN_MODEPLUS  "a+": 	Opens for reading and appending; the appending operation includes the removal of the EOF marker before new data is written to the file and the EOF marker is restored after writing is complete; creates the file first if it doesn’t exist.
																															When a file is opened with the "a" or "a+" access type, all write operations occur at the end of the file. The file pointer can be repositioned using FB_FileSeek, but is always moved back to the end of the file before any write operation is carried out. Thus, existing data cannot be overwritten. 																				                                    								
																				FOPEN_MODEBINARY  "b": Open in binary (untranslated) mode.
																				FOPEN_MODETEXT  "t": Open in text (translated) mode. *)
	Path													:	T_MaxString; // \\PC-Name\Folder\ 
	FileName												:	T_MaxString := ''; // NewFile.xyz 
	OldFileName												:	T_MaxString := ''; // File.xyz 
	pBuffer													:	PVOID; //pointer to data section 
	Length													: 	UDINT; // sizeof data section for read and write. Note to use "LEN" while writing-command, beacause otherwise the whole datasection and not only the string will be written 
	SeekOrigin												: 	E_SeekOrigin := SEEK_SET; //Seek function parameter - Contains the relative position for the move.
	SeekPos													:	DINT; //Seek function parameter - Contains the desired (new) target position of the file pointer.
END_VAR
VAR_OUTPUT
	EOF														:	BOOL;	//This output is switched to TRUE if the end of file is reached.
	WorkedLen												:	UDINT;	//Contains the number of bytes currently read or written
	hFile													:	UINT;	//File handle of currently opened file
	ActSeekPos												:	DINT;	//Act file pointer position of filled by Tell function
	Line   													: T_MaxString; //Read line of file - filled by function Gets

END_VAR
VAR
(* internal used variables ************************************************************)
	MemErrorText											:	STRING(50);
	MemFnc													:	INT := -1;
	
(* trigger ******************************************************************************)

(* function-block instances ************************************************************)
	File_Open												:	FB_FileOpen;
	File_Close												: 	FB_FileClose;
	File_Read 												: 	FB_FileRead;
	File_Write												:	FB_FileWrite;
	File_Delete												:	FB_FileDelete;
	File_Rename												:	FB_FileRename;
	File_Puts												:	FB_FilePuts;
	File_Gets												:	FB_FileGets;
	File_CreateDir											:	FB_CreateDir;
	File_RemoveDir											:	FB_RemoveDir;
	File_Tell												:	FB_FileTell ;
	File_Seek												:	FB_FileSeek ;
	File_EoF												:	FB_EOF;
END_VAR

	(* FileHandling												V2.0	*)
	(********************************************************************)

(* Sequence **********************************************************************)
	rtExecute(CLK := Execute);
	IF rtExecute.Q
		AND MemFnc < 0
	THEN
		Busy												:= TRUE;
		Done												:= FALSE;
		Error												:= FALSE;
		ErrorId												:= 0;
		CASE fnc OF                     					
		FNC_OPEN:		MemFnc 								:= fnc;
		FNC_READ:		MemFnc 								:= fnc;
		FNC_WRITE:		MemFnc 								:= fnc;
		FNC_PUTS:		MemFnc 								:= fnc;
		FNC_GETS:		MemFnc 								:= fnc;
		FNC_CLOSE:		MemFnc 								:= fnc;
		FNC_DELETE:		MemFnc 								:= fnc;
		FNC_RENAME:		MemFnc 								:= fnc;
		FNC_REMOVEDIR: 	MemFnc 								:= fnc;
		FNC_CREATEDIR: 	MemFnc 								:= fnc;
		FNC_SEEK:		MemFnc 								:= fnc;
		FNC_TELL:		MemFnc 								:= fnc;
		FNC_EOF:		MemFnc 								:= fnc;
		ELSE                            					
			ErrorId											:= E_AdsErr.DEVICE_INVALIDPARM;
			Error											:= TRUE;
			Done											:= FALSE;
			Busy											:= FALSE;
		END_CASE
	END_IF

	CASE MemFnc OF
		FNC_OPEN:		Open(Execute := Execute);
		FNC_READ:		Read(Execute := Execute);
		FNC_WRITE:		Write(Execute := Execute);
		FNC_PUTS:		Puts(Execute := Execute);
		FNC_GETS:		Gets(Execute := Execute);
		FNC_CLOSE:		Close(Execute := Execute);
		FNC_DELETE:		Delete(Execute := Execute);
		FNC_RENAME:		Rename(Execute := Execute);
		FNC_REMOVEDIR: 	RemoveDir(Execute := Execute);
		FNC_CREATEDIR: 	CreateDir(Execute := Execute);
		FNC_SEEK:		Seek(Execute := Execute);
		FNC_TELL:		Tell(Execute := Execute);
		FNC_EOF:		IsEof(Execute := Execute);
	
	-1:
		IF NOT Execute
		THEN
			Busy											:= FALSE;
			Done											:= FALSE;
			Error											:= FALSE;
			ErrorID											:= 0;
		END_IF
	END_CASE
(*************************************************************************)

METHOD PUBLIC close : Bool //Return value = TRUE if busy
VAR_INPUT
	Execute		:	BOOL	:= FALSE;
END_VAR
	IF Execute
	THEN
		Error												:=	FALSE;
		ErrorId												:= 0;
		File_Close.bExecute 								:= TRUE;
	ELSIF NOT File_Close.bBusy      						
	THEN                            						
		Error												:=	FALSE;
		ErrorId												:= 0;
		File_Close.bExecute 								:= FALSE;
	END_IF                          						
                                    	
	MemFnc 													:= FNC_CLOSE;
	THIS^.Execute											:= Execute;

	File_Close(
		sNetId		:= AMSNetId,
		hFile		:= hFile,
		bExecute	:= ,
		tTimeout	:= Timeout,
		bBusy		=> Busy,
		bError		=> ,
		nErrId		=> );

	IF NOT File_Close.bBusy
		AND NOT File_Close.bError
		AND File_Close.bExecute
	THEN
		Done												:= TRUE;
		hFile 												:= 0;
	ELSE                            						
		Done												:= FALSE;
	END_IF

	IF NOT Busy
	THEN
		IF File_Close.bExecute
		THEN
			Error											:=	File_Close.bError;
			ErrorId											:= File_Close.nErrId;
		END_IF
		IF NOT Execute
		THEN
			MemFnc											:=  -1;
			File_Close(bExecute 							:= FALSE);
		END_IF
	END_IF

	(* Fehler speichern *)
	IF Error
	THEN
		MemErrorText										:= CONCAT('File_Close ErrorID: ', UDINT_TO_STRING(ErrorID));
	END_IF
	
	Close													:= Busy;
END_METHOD

METHOD PUBLIC createDir : BOOL //Return value = TRUE if busy
//required parameter
//Path
VAR_INPUT
	Execute													:	BOOL;
END_VAR
	IF Execute
	THEN
		Error												:=	FALSE;
		ErrorId												:= 0;
		File_CreateDir.bExecute 							:= TRUE;
	ELSIF NOT File_CreateDir.bBusy      					
	THEN                                					
		Error												:=	FALSE;
		ErrorId												:= 0;
		File_CreateDir.bExecute								:= FALSE;
	END_IF                              					
                                        	
	MemFnc 													:= FNC_CREATEDIR;
	THIS^.Execute											:= Execute;

	File_CreateDir(
		sNetId		:= AMSNetId,
		sPathName	:= Path,
		ePath		:= ,
		bExecute	:= ,
		tTimeout	:= Timeout,
		bBusy		=> Busy,
		bError		=> ,
		nErrId		=> );

	Done													:= NOT File_CreateDir.bBusy
																AND NOT File_CreateDir.bError
																AND File_CreateDir.bExecute;
	IF NOT Busy
	THEN
		IF File_CreateDir.bExecute
		THEN
			Error											:=	File_CreateDir.bError;
			ErrorId											:= File_CreateDir.nErrId;
		END_IF
		IF NOT Execute
		THEN
			MemFnc											:=  -1;
			File_CreateDir(bExecute := FALSE);
		END_IF
	END_IF


	IF Error
	THEN
		MemErrorText										:= CONCAT('File_CreateDir ErrorID: ', UDINT_TO_STRING(ErrorID));
	END_IF
	
	CreateDir												:= Busy;
END_METHOD

METHOD PUBLIC delete : BOOL //Return value = TRUE if busy
//required parameter
//Path
//FileName
VAR_INPUT
	Execute			:	bool;
END_VAR
	IF Execute
	THEN
		Error												:=	FALSE;
		ErrorId												:= 0;
		File_Delete.bExecute 								:= TRUE;
	ELSIF NOT File_Delete.bBusy         					
	THEN                                					
		Error												:=	FALSE;
		ErrorId												:= 0;
		File_Delete.bExecute 								:= FALSE;
	END_IF                              					
                                        	
	MemFnc 													:= FNC_DELETE;
	THIS^.Execute											:= Execute;

	File_Delete(
		sNetId		:= AMSNetId,
		sPathName	:= CONCAT(Path,FileName),
		ePath		:= ,
		bExecute	:= ,
		tTimeout	:= Timeout,
		bBusy		=> Busy,
		bError		=> ,
		nErrId		=> );

	Done													:= 	NOT File_Delete.bBusy
																AND NOT File_Delete.bError
																AND File_Delete.bExecute;
	IF NOT Busy
	THEN
		IF File_Delete.bExecute
		THEN
			Error											:=	File_Delete.bError;
			ErrorId											:= File_Delete.nErrId;
		END_IF
		IF NOT Execute
		THEN
			MemFnc											:= -1;
			File_Delete(bExecute := FALSE);
		END_IF
	END_IF


	IF Error
	THEN
		MemErrorText										:= CONCAT('File_Delete ErrorID: ', UDINT_TO_STRING(ErrorID));
	End_if
	
	Delete													:= Busy;
END_METHOD

METHOD PUBLIC gets : BOOL //Return value = TRUE if busy
//required parameter
//Path
//Filename
//Mode
//pBuffer
VAR_INPUT
	Execute			:	BOOL;
END_VAR
IF pBuffer = 0 THEN
	Busy													:= NOT Error;
	Error													:= TRUE;
	ErrorId													:= E_AdsErr.DEVICE_INVALIDPARM;
	Done													:= FALSE;
	MemFnc													:= -1 ;
	RETURN;                             					
END_IF                                  					
                                        					
	MemFnc 													:= FNC_GETS;
	THIS^.Execute											:= Execute;
                                        					
	CASE State OF                       	
	0:                                  	
		IF Execute                      	
		THEN                            	
			Done											:= FALSE;
			Error											:= FALSE;
			ErrorId 										:= 0;
			
			File_Open(bExecute := FALSE);
			File_Gets(bExecute := FALSE);
			File_Close(bExecute := FALSE);
			
			EOF												:= FALSE;
			WorkedLen										:= 0;
			
			IF hFile = 0
			THEN
				File_Open(
					sNetId		:= AMSNetId,
					sPathName	:= CONCAT(Path,FileName),
					nMode		:= Mode ,
					ePath		:= (* Default *),
					bExecute	:= TRUE,
					tTimeout	:= Timeout,
					bBusy		=> ,
					bError		=> ,
					nErrId		=> ,
					hFile		=> );

				State 										:= 10;
			ELSE                							
				State 										:= 10;
			END_IF
		ELSE
			Done											:= FALSE;
			Error											:= FALSE;
			ErrorId 										:= 0;
		END_IF

	10:
		File_Open();

		IF NOT File_Open.bBusy
		THEN
			IF File_Open.bError
			THEN
				State 										:= 99;
			ELSE
				IF File_Open.bExecute THEN hFile := File_Open.hFile; END_IF
				File_Gets(
					sNetId		:= AMSNetId,
					hFile		:= hFile,
					bExecute	:= TRUE,
					tTimeout	:= Timeout,
					sLine		=> ,
					bEOF		=> ,
					bBusy		=> ,
					bError		=> ,
					nErrId		=> );

				State 										:= 20;
			END_IF
		END_IF

	20:
		File_Gets(bEOF		=> EOF);
		IF NOT File_Gets.bBusy
		THEN
			IF NOT File_Gets.bError
			THEN
				IF pBuffer <> 0 AND Length <> 0
				THEN
					 MEMCPY(pBuffer , ADR(File_Gets.sLine), MIN(TO_UDINT(Length), SIZEOF(File_Gets.sLine)));
				END_IF
				Line										:= File_Gets.sLine;
			END_IF
			IF File_Open.bExecute
			THEN
				File_Close(
					sNetId	:= AMSNetId,
					hFile	:= hFile,
					bExecute:= TRUE,
					tTimeout:= Timeout,
					bBusy	=> ,
					bError	=> ,
					nErrId	=> );
				State										:= 30;
			ELSE
				State										:= 99;
			END_IF

		END_IF

	30:
		File_Close();
		IF NOT File_Close.bBusy
		THEN
			hFile											:= 0;
			State											:= 99;
		END_IF

	99:
		IF NOT Execute
		THEN
			Memfnc											:= -1;
			state 											:= 0;
		END_IF
	END_CASE

	Done													:= state = 99
																AND NOT File_Gets.bError
																AND NOT File_Close.bError
																AND NOT File_Open.bError;
                                        					
	Error													:= state = 99
																AND(
																File_Gets.bError
																OR File_Close.bError
																OR File_Open.bError);
                                        					
	Busy													:= state <> 0
																AND NOT Done
																AND NOT Error;

	IF Error
	THEN
		IF File_Close.bError 	THEN 	ErrorId :=  File_Close.nErrId; 	END_IF
		IF File_Gets.bError 	THEN 	ErrorId :=  File_Gets.nErrId; 	END_IF
		IF File_Open.bError 	THEN	ErrorId :=  File_Open.nErrId; 	END_IF
	ELSE
		ErrorId 											:= 0;
	END_IF                              					
                                        					
	IF NOT Execute                      					
		AND state = 99                  					
	THEN                                					
			MemFnc											:= -1;
		state 												:= 0;
	END_IF                              	
                                        	
	IF Error                            	
	THEN                                	
		MemErrorText										:= CONCAT('File_Gets ErrorID: ', UDINT_TO_STRING(ErrorID));
	END_IF                              					
                                        					
	Gets													:= Busy;
END_METHOD

METHOD PUBLIC isEoF : BOOL //Return value = TRUE if busy
VAR_INPUT
	Execute													:	BOOL;
END_VAR
	IF Execute
	THEN
		Error												:=	FALSE;
		ErrorId												:= 0;
		File_EoF.bExecute 									:= TRUE;
	ELSIF NOT File_EoF.bBusy           					
	THEN                                					
		Error												:=	FALSE;
		ErrorId												:= 0;
		File_EoF.bExecute 									:= FALSE;
	END_IF                              							
	                                    	
	MemFnc 													:= FNC_EOF;
	THIS^.Execute											:= Execute;
                                        	
	File_EoF(
		sNetId		:= AMSNetId,
		hFile		:= hFile ,
		tTimeout	:= Timeout,
		bBusy		=> Busy,
		bError		=> ,
		nErrId		=> ,
		bEoF		=> EoF);

	Done													:= NOT File_EoF.bBusy
																AND NOT File_EoF.bError
																AND File_EoF.bExecute;
	IF NOT Busy                         					
	THEN                        					
		IF File_EoF.bExecute           					
		THEN                            	
			Error											:=	File_EoF.bError;
			ErrorId											:= File_EoF.nErrId;
		END_IF
		IF NOT Execute
		THEN
			MemFnc											:= 1;
			File_EoF(bExecute := FALSE);
		END_IF
	END_IF


	IF Error
	THEN
		MemErrorText										:= CONCAT('File_EoF ErrorID: ', UDINT_TO_STRING(ErrorID));
	END_IF
	
	IsEoF													:= Busy;
END_METHOD

METHOD PUBLIC open : BOOL //Return value = TRUE if busy
//required parameter
//Path
//FileName
//Mode
VAR_INPUT
	Execute				:	BOOL; 
END_VAR
IF Execute
THEN
	Error													:= FALSE;
	ErrorId													:= 0;
	File_Open.bExecute 										:= TRUE;
ELSIF NOT File_Open.bBusy           						
THEN                                						
	Error													:=	FALSE;
	ErrorId													:= 0;
	File_Open.bExecute 										:= FALSE;
END_IF	

MemFnc 														:= FNC_OPEN;
THIS^.Execute												:= Execute;

(* Work File Open *)
File_Open(
	sNetId		:= AMSNetId,
	sPathName	:= CONCAT(Path,FileName),
	nMode		:= Mode ,
	ePath		:= (* Default *),
	bExecute	:= ,
	tTimeout	:= Timeout,
	bBusy		=> Busy,
	bError		=> ,
	nErrId		=> ,
	hFile		=> hFile);

Done														:= NOT File_Open.bBusy
																AND NOT File_Open.bError
																AND File_Open.bExecute;
IF NOT Busy
THEN
	IF File_Open.bExecute
	THEN
		Error												:=	File_Open.bError;
		ErrorId												:= File_Open.nErrId;
	END_IF
	IF NOT Execute
	THEN
		MemFnc												:= -1;
		File_Open(bExecute := FALSE);
	END_IF
END_IF

IF Error
THEN
	MemErrorText											:= CONCAT('File_Open ErrorID: ', UDINT_TO_STRING(ErrorID));
END_IF                              						
                                    	
Open														:= Busy;
END_METHOD

METHOD PUBLIC puts : BOOL //Return value = TRUE if busy
//required parameter
//Path
//FileName
//Mode
//pBuffer
//Lenght
VAR_INPUT
	Execute				:	BOOL;
END_VAR
IF pBuffer = 0 THEN
	Busy													:= NOT Error;
	Error													:= TRUE;
	ErrorId													:= E_AdsErr.DEVICE_INVALIDPARM;
	Done													:= FALSE;
	MemFnc													:= -1 ;
	RETURN;
END_IF

	MemFnc 													:= FNC_PUTS;
	THIS^.Execute											:= Execute;

	CASE State OF
	0:
		IF Execute
		THEN
			Done											:= FALSE;
			Error											:= FALSE;
			ErrorId 										:= 0;
			
			File_Open(bExecute := FALSE);
			File_Puts(bExecute := FALSE);
			File_Close(bExecute := FALSE);
			
			EOF												:= FALSE;
			WorkedLen										:= 0;
			
			IF hFile = 0
			THEN
				File_Open(
					sNetId		:= AMSNetId,
					sPathName	:= CONCAT(Path,FileName),
					nMode		:= Mode ,
					ePath		:= (* Default *),
					bExecute	:= TRUE,
					tTimeout	:= Timeout,
					bBusy		=> ,
					bError		=> ,
					nErrId		=> ,
					hFile		=> );

				State 										:= 10;
			ELSE                							
				State 										:= 10;
			END_IF              							
		ELSE                    							
			Done											:= FALSE;
			Error											:= FALSE;
			ErrorId 										:= 0;
		END_IF

	10:
		File_Open();

		IF NOT File_Open.bBusy
		THEN
			IF File_Open.bError
			THEN
				State 										:= 99;
			ELSE
				IF File_Open.bExecute THEN hFile := File_Open.hFile; END_IF
				MEMCPY(ADR(File_Puts.sLine),  pBuffer, MIN(TO_UDINT(Length), SIZEOF(File_Puts.sLine)));
				File_Puts(
					sNetId		:= AMSNetId,
					hFile		:= hFile,
					sLine		:= (* siehe oben *),
					bExecute	:= TRUE,
					tTimeout	:= Timeout,
					bBusy		=> ,
					bError		=> ,
					nErrId		=> );

				State 										:= 20;
			END_IF
		END_IF

	20:
		MEMCPY(ADR(File_Puts.sLine),  pBuffer, MIN(TO_UDINT(Length), SIZEOF(File_Puts.sLine)));
		File_Puts();

		IF NOT File_Puts.bBusy
		THEN
			IF File_Open.bExecute
			THEN
				File_Close(
					sNetId	:= AMSNetId,
					hFile	:= hFile,
					bExecute:= TRUE,
					tTimeout:= Timeout,
					bBusy	=> ,
					bError	=> ,
					nErrId	=> );
				State										:= 30;
			ELSE
				State										:= 99;
			END_IF

		END_IF

	30:
		File_Close();
		IF NOT File_Close.bBusy
		THEN
			hFile						:= 0;
			State						:= 99;
		END_IF

	99:
		IF NOT Execute
		THEN
			Memfnc					:= -1;
			state 					:= 0;
		END_IF
	END_CASE

	Done							:= state = 99
										AND NOT File_Puts.bError
										AND NOT File_Close.bError
										AND NOT File_Open.bError;

	Error							:= state = 99
										AND(
										File_Puts.bError
										OR File_Close.bError
										OR File_Open.bError);

	Busy							:= state <> 0
										AND NOT Done
										AND NOT Error;

	IF Error
	THEN
		IF File_Close.bError 	THEN	ErrorId :=  File_Close.nErrId; 	END_IF
		IF File_Puts.bError 	THEN 	ErrorId :=  File_Puts.nErrId; 	END_IF
		IF File_Open.bError 	THEN 	ErrorId :=  File_Open.nErrId;	END_IF
	ELSE
		ErrorId 					:= 0;
	END_IF

	IF NOT Execute
		AND state = 99
	THEN
		MemFnc						:= -1;
		state 						:= 0;
	END_IF

	IF Error
	THEN
		MemErrorText				:= CONCAT('File_Puts ErrorID: ', UDINT_TO_STRING(ErrorID));
	END_IF
	
	Puts							:= Busy;
END_METHOD

METHOD PUBLIC read : BOOL //Return value = TRUE if busy
//required parameter
//Path
//FileName
//Mode
//pBuffer
//Lenght
VAR_INPUT
	Execute			:	BOOL;
END_VAR
IF pBuffer = 0 THEN
	Busy													:= NOT Error;
	Error													:= TRUE;
	ErrorId													:= E_AdsErr.DEVICE_INVALIDPARM;
	Done													:= FALSE;
	MemFnc													:= -1 ;
	RETURN;                             					
END_IF                                  					
                                        	
	MemFnc 													:= FNC_READ;
	THIS^.Execute											:= Execute;

	CASE State OF
	0:
		IF Execute
		THEN
			Done											:= FALSE;
			Error											:= FALSE;
			ErrorId 										:= 0;
			
			File_Open(bExecute := FALSE);
			File_Read(bExecute := FALSE);
			File_Close(bExecute := FALSE);
			
			EOF												:= FALSE;
			WorkedLen										:= 0;
			
			IF hFile = 0
			THEN
				File_Open(
					sNetId		:= AMSNetId,
					sPathName	:= CONCAT(Path,FileName),
					nMode		:= Mode ,
					ePath		:= (* Default *),
					bExecute	:= TRUE,
					tTimeout	:= Timeout,
					bBusy		=> ,
					bError		=> ,
					nErrId		=> ,
					hFile		=> );

				State 										:= 10;
			ELSE                    						
				State 										:= 10;
			END_IF                  						
		ELSE                        						
			Done											:= FALSE;
			Error											:= FALSE;
			ErrorId 										:= 0;
		END_IF

	10:
		File_Open();
		IF NOT File_Open.bBusy
		THEN
			IF File_Open.bError
			THEN
				State 										:= 99;
			ELSE
				IF File_Open.bExecute THEN hFile := File_Open.hFile; END_IF
				File_Read(
					sNetId		:= AmsNetId,
					hFile		:= hFile,
					pReadBuff	:= pBuffer,
					cbReadLen	:= Length,
					bExecute	:= TRUE,
					tTimeout	:= Timeout,
					bBusy		=> ,
					bError		=> ,
					nErrId		=> ,
					cbRead		=> ,
					bEOF		=> );

				State 										:= 20;
			END_IF
		END_IF

	20:
		File_Read(
			pReadBuff	:= pBuffer,
			cbReadLen	:= Length,
			bExecute	:= TRUE,
			cbRead		=> WorkedLen,
			bEOF		=> EOF);

		IF NOT File_Read.bBusy
		THEN
			IF File_Open.bExecute
			THEN
				File_Close(
					sNetId	:= AMSNetId,
					hFile	:= hFile,
					bExecute:= TRUE,
					tTimeout:= Timeout,
					bBusy	=> ,
					bError	=> ,
					nErrId	=> );
				State										:= 30;
			ELSE                        						
				State										:= 99;
			END_IF                      						
                                        						
		END_IF                          						
                                        						
	30:                                 						
		File_Close();                   						
		IF NOT File_Close.bBusy         						
		THEN                            						
			hFile											:= 0;
			State											:= 99;
		END_IF                          						
                                        						
	99:                                 						
		IF NOT Execute                  						
		THEN                            				
			Memfnc											:= -1;
			state 											:= 0;
		END_IF                          	
	END_CASE                            	
                                        	
	Done													:= state = 99
																AND NOT File_Read.bError
																AND NOT File_Close.bError
																AND NOT File_Open.bError;
	                                    						
	Error													:= state = 99
																AND(
																File_Read.bError
																OR File_Close.bError
																OR File_Open.bError);
	                                    						
	Busy													:= state <> 0
																AND NOT Done
																AND NOT Error;

	IF Error
	THEN
		IF File_Close.bError	THEN 	ErrorId :=  File_Close.nErrId;	END_IF
		IF File_Read.bError 	THEN	ErrorId :=  File_Read.nErrId; 	END_IF
		IF File_Open.bError		THEN	ErrorId :=  File_Open.nErrId; 	END_IF
	ELSE
		ErrorId 											:= 0;
	END_IF                              						
                                        						
